	// Place to Basket 		
	4:
		IF process_Z = 0 THEN
			CASE GVL.Basket_A_Counter OF
				0:
					bit1 					:= 4;
					bit2 					:= 2;
					KR1.bOutBit[ bit1,bit2] := TRUE; //210
					MSG_Bskt				:= MSG.ACTION_FGA_POS1;
					process_Z 				:= 1;
				1:
					bit1 					:= 4;
					bit2 					:= 3;
					KR1.bOutBit[ bit1,bit2] := TRUE; //210
					MSG_Bskt				:= MSG.ACTION_FGA_POS2;
					process_Z 				:= 1;
					RETURN;
				2:
					bit1 					:= 4;
					bit2 					:= 4;
					KR1.bOutBit[ bit1,bit2] := TRUE; //210
					MSG_Bskt				:= MSG.ACTION_FGA_POS3;
					process_Z 				:= 1;
				3:
					bit1 					:= 4;
					bit2 					:= 5;
					KR1.bOutBit[ bit1,bit2] := TRUE; //210
					MSG_Bskt				:= MSG.ACTION_FGA_POS4;
					process_Z 				:= 1;
				4:
					bit1 					:= 4;
					bit2 					:= 6;
					KR1.bOutBit[ bit1,bit2] := TRUE; //210
					MSG_Bskt				:= MSG.ACTION_FGA_POS5;
					process_Z 				:= 1;
				5:
					bit1 					:= 4;
					bit2 					:= 7;
					KR1.bOutBit[ bit1,bit2] := TRUE; //210
					MSG_Bskt				:= MSG.ACTION_FGA_POS6;
					process_Z 				:= 1;
				6:
					bit1 					:= 5;
					bit2 					:= 0;
					KR1.bOutBit[ bit1,bit2] := TRUE; //210
					MSG_Bskt				:= MSG.ACTION_FGA_POS7;
					process_Z 				:= 1;
				7:
					bit1 					:= 5;
					bit2 					:= 1;
					KR1.bOutBit[ bit1,bit2] := TRUE; //210
					MSG_Bskt				:= MSG.ACTION_FGA_POS8;
					process_Z 				:= 1;
				8:
					bit1 					:= 5;
					bit2 					:= 2;
					KR1.bOutBit[ bit1,bit2] := TRUE; //210
					MSG_Bskt				:= MSG.ACTION_FGA_POS9;
					process_Z 				:= 1;
				9:
					bit1 					:= 5;
					bit2 					:= 3;
					KR1.bOutBit[ bit1,bit2] := TRUE; //210
					MSG_Bskt				:= MSG.ACTION_FGA_POS10;
					process_Z 				:= 1;
				10:
					bit1 					:= 5;
					bit2 					:= 4;
					KR1.bOutBit[ bit1,bit2] := TRUE; //210
					MSG_Bskt				:= MSG.ACTION_FGA_POS11;
					process_Z 				:= 1;
				11:
					bit1 					:= 5;
					bit2 					:= 5;
					KR1.bOutBit[ bit1,bit2] := TRUE; //210
					MSG_Bskt				:= MSG.ACTION_FGA_POS12;
					process_Z 				:= 1;
				12:
					bit1 					:= 5;
					bit2 					:= 6;
					KR1.bOutBit[ bit1,bit2] := TRUE; //210
					MSG_Bskt				:= MSG.ACTION_FGA_POS13;
					process_Z 				:= 1;
				13:
					bit1 					:= 5;
					bit2 					:= 7;
					KR1.bOutBit[ bit1,bit2] := TRUE; //210
					MSG_Bskt				:= MSG.ACTION_FGA_POS14;
					process_Z 				:= 1;
				14:
					bit1 					:= 6;
					bit2 					:= 0;
					KR1.bOutBit[ bit1,bit2] := TRUE; //210
					MSG_Bskt				:= MSG.ACTION_FGA_POS15;
					process_Z 				:= 1;
				15:
					bit1 					:= 6;
					bit2 					:= 1;
					KR1.bOutBit[ bit1,bit2] := TRUE; //210
					MSG_Bskt				:= MSG.ACTION_FGA_POS16;
					process_Z 				:= 1;
				16:
					bit1 					:= 6;
					bit2 					:= 2;
					KR1.bOutBit[ bit1,bit2] := TRUE; //210
					MSG_Bskt				:= MSG.ACTION_FGA_POS17;
					process_Z 				:= 1;
				17:
					bit1 					:= 6;
					bit2 					:= 3;
					KR1.bOutBit[ bit1,bit2] := TRUE; //210
					MSG_Bskt				:= MSG.ACTION_FGA_POS18;
					process_Z 				:= 1;
				18:
					bit1 					:= 6;
					bit2 					:= 4;
					KR1.bOutBit[ bit1,bit2] := TRUE; //210
					MSG_Bskt				:= MSG.ACTION_FGA_POS19;
					process_Z 				:= 1;
				19:
					bit1 					:= 6;
					bit2 					:= 5;
					KR1.bOutBit[ bit1,bit2] := TRUE; //210
					MSG_Bskt				:= MSG.ACTION_FGA_POS20;
					process_Z 				:= 1;
				20:
					bit1 					:= 6;
					bit2 					:= 6;
					KR1.bOutBit[ bit1,bit2] := TRUE; //210
					MSG_Bskt				:= MSG.ACTION_FGA_POS21;
					process_Z 				:= 1;
				21:
					bit1 					:= 6;
					bit2 					:= 7;
					KR1.bOutBit[ bit1,bit2] := TRUE; //210
					MSG_Bskt				:= MSG.ACTION_FGA_POS22;
					process_Z 				:= 1;
				22:
					bit1 					:= 7;
					bit2 					:= 0;
					KR1.bOutBit[ bit1,bit2] := TRUE; //210
					MSG_Bskt				:= MSG.ACTION_FGA_POS23;
					process_Z 				:= 1;
				23:
					bit1 					:= 7;
					bit2 					:= 1;
					KR1.bOutBit[ bit1,bit2] := TRUE; //210
					MSG_Bskt				:= MSG.ACTION_FGA_POS24;
					process_Z 				:= 1;
				24:
					bit1 					:= 7;
					bit2 					:= 2;
					KR1.bOutBit[ bit1,bit2] := TRUE; //210
					MSG_Bskt				:= MSG.ACTION_FGA_POS25;
					process_Z 				:= 1;
				25:
					bit1 					:= 7;
					bit2 					:= 3;
					KR1.bOutBit[ bit1,bit2] := TRUE; //210
					MSG_Bskt				:= MSG.ACTION_FGA_POS26;
					process_Z 				:= 1;
				26:
					bit1 					:= 7;
					bit2 					:= 4;
					KR1.bOutBit[ bit1,bit2] := TRUE; //210
					MSG_Bskt				:= MSG.ACTION_FGA_POS27;
					process_Z 				:= 1;
				27:
					bit1 					:= 7;
					bit2 					:= 5;
					KR1.bOutBit[ bit1,bit2] := TRUE; //210
					MSG_Bskt				:= MSG.ACTION_FGA_POS28;
					process_Z 				:= 1;
				28:
					bit1 					:= 7;
					bit2 					:= 6;
					KR1.bOutBit[ bit1,bit2] := TRUE; //210
					MSG_Bskt				:= MSG.ACTION_FGA_POS29;
					process_Z 				:= 1;
				29:
					bit1 					:= 7;
					bit2 					:= 7;
					KR1.bOutBit[ bit1,bit2] := TRUE; //210
					MSG_Bskt				:= MSG.ACTION_FGA_POS30;
					process_Z 				:= 1;
				30:
					bit1 					:= 8;
					bit2 					:= 0;
					KR1.bOutBit[ bit1,bit2] := TRUE; //210
					MSG_Bskt				:= MSG.ACTION_FGA_POS31;
					process_Z 				:= 1;
				31:
					bit1 					:= 8;
					bit2 					:= 1;
					KR1.bOutBit[ bit1,bit2] := TRUE; //210
					MSG_Bskt				:= MSG.ACTION_FGA_POS32;
					process_Z 				:= 1;
				32:
					bit1 					:= 8;
					bit2 					:= 2;
					KR1.bOutBit[ bit1,bit2] := TRUE; //210
					MSG_Bskt				:= MSG.ACTION_FGA_POS33;
					process_Z 				:= 1;
				33:
					bit1 					:= 8;
					bit2 					:= 3;
					KR1.bOutBit[ bit1,bit2] := TRUE; //210
					MSG_Bskt				:= MSG.ACTION_FGA_POS34;
					process_Z 				:= 1;
				34:
					bit1 					:= 8;
					bit2 					:= 4;
					KR1.bOutBit[ bit1,bit2] := TRUE; //210
					MSG_Bskt				:= MSG.ACTION_FGA_POS35;
					process_Z 				:= 1;
				35:
					bit1 					:= 8;
					bit2 					:= 5;
					KR1.bOutBit[ bit1,bit2] := TRUE; //210
					MSG_Bskt				:= MSG.ACTION_FGA_POS36;
					process_Z 				:= 1;
				36:
					bit1 					:= 8;
					bit2 					:= 6;
					KR1.bOutBit[ bit1,bit2] := TRUE; //210
					MSG_Bskt				:= MSG.ACTION_FGA_POS37;
					process_Z 				:= 1;
				37:
					bit1 					:= 8;
					bit2 					:= 7;
					KR1.bOutBit[ bit1,bit2] := TRUE; //210
					MSG_Bskt				:= MSG.ACTION_FGA_POS38;
					process_Z 				:= 1;
				38:
					bit1 					:= 9;
					bit2 					:= 0;
					KR1.bOutBit[ bit1,bit2] := TRUE; //210
					MSG_Bskt				:= MSG.ACTION_FGA_POS39;
					process_Z 				:= 1;
				39:
					bit1 					:= 9;
					bit2 					:= 1;
					KR1.bOutBit[ bit1,bit2] := TRUE; //210
					MSG_Bskt				:= MSG.ACTION_FGA_POS40;
					process_Z 				:= 1;
				40:
					bit1 					:= 9;
					bit2 					:= 2;
					KR1.bOutBit[ bit1,bit2] := TRUE; //210
					MSG_Bskt				:= MSG.ACTION_FGA_POS41;
					process_Z 				:= 1;
				41:
					bit1 					:= 9;
					bit2 					:= 3;
					KR1.bOutBit[ bit1,bit2] := TRUE; //210
					MSG_Bskt				:= MSG.ACTION_FGA_POS42;
					process_Z 				:= 1;
				42:
					bit1 					:= 9;
					bit2 					:= 4;
					KR1.bOutBit[ bit1,bit2] := TRUE; //210
					MSG_Bskt				:= MSG.ACTION_FGA_POS43;
					process_Z 				:= 1;
				43:
					bit1 					:= 9;
					bit2 					:= 5;
					KR1.bOutBit[ bit1,bit2] := TRUE; //210
					MSG_Bskt				:= MSG.ACTION_FGA_POS44;
					process_Z 				:= 1;
				44:
					bit1 					:= 9;
					bit2 					:= 6;
					KR1.bOutBit[ bit1,bit2] := TRUE; //210
					MSG_Bskt				:= MSG.ACTION_FGA_POS45;
					process_Z 				:= 1;
				45:
					bit1 					:= 9;
					bit2 					:= 7;
					KR1.bOutBit[ bit1,bit2] := TRUE; //210
					MSG_Bskt				:= MSG.ACTION_FGA_POS46;
					process_Z 				:= 1;
				46:
					bit1 					:= 10;
					bit2 					:= 0;
					KR1.bOutBit[ bit1,bit2] := TRUE; //210
					MSG_Bskt				:= MSG.ACTION_FGA_POS47;
					process_Z 				:= 1;
				47:
					bit1 					:= 10;
					bit2 					:= 1;
					KR1.bOutBit[ bit1,bit2] := TRUE; //210
					MSG_Bskt				:= MSG.ACTION_FGA_POS48;
					process_Z 				:= 1;
				48:
					bit1 					:= 10;
					bit2 					:= 2;
					KR1.bOutBit[ bit1,bit2] := TRUE; //210
					MSG_Bskt				:= MSG.ACTION_FGA_POS49;
					process_Z 				:= 1;
				49:
					bit1 					:= 10;
					bit2 					:= 3;
					KR1.bOutBit[ bit1,bit2] := TRUE; //210
					MSG_Bskt				:= MSG.ACTION_FGA_POS50;
					process_Z 				:= 1;
				50:
					bit1 					:= 10;
					bit2 					:= 4;
					KR1.bOutBit[ bit1,bit2] := TRUE; //210
					MSG_Bskt				:= MSG.ACTION_FGA_POS51;
					process_Z 				:= 1;
				51:
					bit1 					:= 10;
					bit2 					:= 5;
					KR1.bOutBit[ bit1,bit2] := TRUE; //210
					MSG_Bskt				:= MSG.ACTION_FGA_POS52;
					process_Z 				:= 1;
				52:
					bit1 					:= 10;
					bit2 					:= 6;
					KR1.bOutBit[ bit1,bit2] := TRUE; //210
					MSG_Bskt				:= MSG.ACTION_FGA_POS53;
					process_Z 				:= 1;
				53:
					bit1 					:= 10;
					bit2 					:= 7;
					KR1.bOutBit[ bit1,bit2] := TRUE; //210
					MSG_Bskt				:= MSG.ACTION_FGA_POS54;
					process_Z 				:= 1;
				54:
					bit1 					:= 11;
					bit2 					:= 0;
					KR1.bOutBit[ bit1,bit2] := TRUE; //210
					MSG_Bskt				:= MSG.ACTION_FGA_POS55;
					process_Z 				:= 1;
				55:
					bit1 					:= 11;
					bit2 					:= 1;
					KR1.bOutBit[ bit1,bit2] := TRUE; //210
					MSG_Bskt				:= MSG.ACTION_FGA_POS56;
					process_Z 				:= 1;
				56:
					bit1 					:= 11;
					bit2 					:= 2;
					KR1.bOutBit[ bit1,bit2] := TRUE; //210
					MSG_Bskt				:= MSG.ACTION_FGA_POS57;
					process_Z 				:= 1;
				57:
					bit1 					:= 11;
					bit2 					:= 3;
					KR1.bOutBit[ bit1,bit2] := TRUE; //210
					MSG_Bskt				:= MSG.ACTION_FGA_POS58;
					process_Z 				:= 1;
				58:
					bit1 					:= 11;
					bit2 					:= 4;
					KR1.bOutBit[ bit1,bit2] := TRUE; //210
					MSG_Bskt				:= MSG.ACTION_FGA_POS59;
					process_Z 				:= 1;
				59:
					bit1 					:= 11;
					bit2 					:= 5;
					KR1.bOutBit[ bit1,bit2] := TRUE; //210
					MSG_Bskt				:= MSG.ACTION_FGA_POS60;
					process_Z 				:= 1;
				60:
					bit1 					:= 11;
					bit2 					:= 6;
					KR1.bOutBit[ bit1,bit2] := TRUE; //210
					MSG_Bskt				:= MSG.ACTION_FGA_POS61;
					process_Z 				:= 1;
				61:
					bit1 					:= 11;
					bit2 					:= 7;
					KR1.bOutBit[ bit1,bit2] := TRUE; //210
					MSG_Bskt				:= MSG.ACTION_FGA_POS62;
					process_Z 				:= 1;
				62:
					bit1 					:= 12;
					bit2 					:= 0;
					KR1.bOutBit[ bit1,bit2] := TRUE; //210
					MSG_Bskt				:= MSG.ACTION_FGA_POS63;
					process_Z 				:= 1;
				63:
					bit1 					:= 12;
					bit2 					:= 1;
					KR1.bOutBit[ bit1,bit2] := TRUE; //210
					MSG_Bskt				:= MSG.ACTION_FGA_POS64;
					process_Z 				:= 1;
				64:
					bit1 					:= 12;
					bit2 					:= 2;
					KR1.bOutBit[ bit1,bit2] := TRUE; //210
					MSG_Bskt				:= MSG.ACTION_FGA_POS65;
					process_Z 				:= 1;
				65:
					bit1 					:= 12;
					bit2 					:= 3;
					KR1.bOutBit[ bit1,bit2] := TRUE; //210
					MSG_Bskt				:= MSG.ACTION_FGA_POS66;
					process_Z 				:= 1;
				66:
					bit1 					:= 12;
					bit2 					:= 4;
					KR1.bOutBit[ bit1,bit2] := TRUE; //210
					MSG_Bskt				:= MSG.ACTION_FGA_POS67;
					process_Z 				:= 1;
				67:
					bit1 					:= 12;
					bit2 					:= 5;
					KR1.bOutBit[ bit1,bit2] := TRUE; //210
					MSG_Bskt				:= MSG.ACTION_FGA_POS68;
					process_Z 				:= 1;
				68:
					bit1 					:= 12;
					bit2 					:= 6;
					KR1.bOutBit[ bit1,bit2] := TRUE; //210
					MSG_Bskt				:= MSG.ACTION_FGA_POS69;
					process_Z 				:= 1;
				69:
					bit1 					:= 12;
					bit2 					:= 7;
					KR1.bOutBit[ bit1,bit2] := TRUE; //210
					MSG_Bskt				:= MSG.ACTION_FGA_POS70;
					process_Z 				:= 1;
				70:
					bit1 					:= 13;
					bit2 					:= 0;
					KR1.bOutBit[ bit1,bit2] := TRUE; //210
					MSG_Bskt				:= MSG.ACTION_FGA_POS71;
					process_Z 				:= 1;
				71:
					bit1 					:= 13;
					bit2 					:= 1;
					KR1.bOutBit[ bit1,bit2] := TRUE; //210
					MSG_Bskt				:= MSG.ACTION_FGA_POS72;
					process_Z 				:= 1;
				72:
					bit1 					:= 13;
					bit2 					:= 2;
					KR1.bOutBit[ bit1,bit2] := TRUE; //210
					MSG_Bskt				:= MSG.ACTION_FGA_POS73;
					process_Z 				:= 1;
				73:
					bit1 					:= 13;
					bit2 					:= 3;
					KR1.bOutBit[ bit1,bit2] := TRUE; //210
					MSG_Bskt				:= MSG.ACTION_FGA_POS74;
					process_Z 				:= 1;
				74:
					bit1 					:= 13;
					bit2 					:= 4;
					KR1.bOutBit[ bit1,bit2] := TRUE; //210
					MSG_Bskt				:= MSG.ACTION_FGA_POS75;
					process_Z 				:= 1;
				75:
					bit1 					:= 13;
					bit2 					:= 5;
					KR1.bOutBit[ bit1,bit2] := TRUE; //210
					MSG_Bskt				:= MSG.ACTION_FGA_POS76;
					process_Z 				:= 1;
				76:
					bit1 					:= 13;
					bit2 					:= 6;
					KR1.bOutBit[ bit1,bit2] := TRUE; //210
					MSG_Bskt				:= MSG.ACTION_FGA_POS77;
					process_Z 				:= 1;
				77:
					bit1 					:= 13;
					bit2 					:= 7;
					KR1.bOutBit[ bit1,bit2] := TRUE; //210
					MSG_Bskt				:= MSG.ACTION_FGA_POS78;
					process_Z 				:= 1;
				78:
					bit1 					:= 14;
					bit2 					:= 0;
					KR1.bOutBit[ bit1,bit2] := TRUE; //210
					MSG_Bskt				:= MSG.ACTION_FGA_POS79;
					process_Z 				:= 1;
				79:
					bit1 					:= 14;
					bit2 					:= 1;
					KR1.bOutBit[ bit1,bit2] := TRUE; //210
					MSG_Bskt				:= MSG.ACTION_FGA_POS80;
					process_Z 				:= 1;
				80:
					bit1 					:= 14;
					bit2 					:= 2;
					KR1.bOutBit[ bit1,bit2] := TRUE; //210
					MSG_Bskt				:= MSG.ACTION_FGA_POS81;
					process_Z 				:= 1;
				81:
					bit1 					:= 14;
					bit2 					:= 3;
					KR1.bOutBit[ bit1,bit2] := TRUE; //210
					MSG_Bskt				:= MSG.ACTION_FGA_POS82;
					process_Z 				:= 1;
				82:
					bit1 					:= 14;
					bit2 					:= 4;
					KR1.bOutBit[ bit1,bit2] := TRUE; //210
					MSG_Bskt				:= MSG.ACTION_FGA_POS83;
					process_Z 				:= 1;
				83:
					bit1 					:= 14;
					bit2 					:= 5;
					KR1.bOutBit[ bit1,bit2] := TRUE; //210
					MSG_Bskt				:= MSG.ACTION_FGA_POS84;
					process_Z 				:= 1;
				84:
					bit1 					:= 14;
					bit2 					:= 6;
					KR1.bOutBit[ bit1,bit2] := TRUE; //210
					MSG_Bskt				:= MSG.ACTION_FGA_POS85;
					process_Z 				:= 1;
				85:
					bit1 					:= 14;
					bit2 					:= 7;
					KR1.bOutBit[ bit1,bit2] := TRUE; //210
					MSG_Bskt				:= MSG.ACTION_FGA_POS86;
					process_Z 				:= 1;
				86:
					bit1 					:= 15;
					bit2 					:= 0;
					KR1.bOutBit[ bit1,bit2] := TRUE; //210
					MSG_Bskt				:= MSG.ACTION_FGA_POS87;
					process_Z 				:= 1;
				87:
					bit1 					:= 15;
					bit2 					:= 1;
					KR1.bOutBit[ bit1,bit2] := TRUE; //210
					MSG_Bskt				:= MSG.ACTION_FGA_POS88;
					process_Z 				:= 1;
				88:
					bit1 					:= 15;
					bit2 					:= 2;
					KR1.bOutBit[ bit1,bit2] := TRUE; //210
					MSG_Bskt				:= MSG.ACTION_FGA_POS89;
					process_Z 				:= 1;
				89:
					bit1 					:= 15;
					bit2 					:= 3;
					KR1.bOutBit[ bit1,bit2] := TRUE; //210
					MSG_Bskt				:= MSG.ACTION_FGA_POS90;
					process_Z 				:= 1;
				90:
					bit1 					:= 15;
					bit2 					:= 4;
					KR1.bOutBit[ bit1,bit2] := TRUE; //210
					MSG_Bskt				:= MSG.ACTION_FGA_POS91;
					process_Z 				:= 1;
				91:
					bit1 					:= 15;
					bit2 					:= 5;
					KR1.bOutBit[ bit1,bit2] := TRUE; //210
					MSG_Bskt				:= MSG.ACTION_FGA_POS92;
					process_Z 				:= 1;
				92:
					bit1 					:= 15;
					bit2 					:= 6;
					KR1.bOutBit[ bit1,bit2] := TRUE; //210
					MSG_Bskt				:= MSG.ACTION_FGA_POS93;
					process_Z 				:= 1;
				93:
					bit1 					:= 15;
					bit2 					:= 7;
					KR1.bOutBit[ bit1,bit2] := TRUE; //210
					MSG_Bskt				:= MSG.ACTION_FGA_POS94;
					process_Z 				:= 1;
				94:
					bit1 					:= 16;
					bit2 					:= 0;
					KR1.bOutBit[ bit1,bit2] := TRUE; //210
					MSG_Bskt				:= MSG.ACTION_FGA_POS95;
					process_Z 				:= 1;
				95:
					bit1 					:= 16;
					bit2 					:= 1;
					KR1.bOutBit[ bit1,bit2] := TRUE; //210
					MSG_Bskt				:= MSG.ACTION_FGA_POS96;
					process_Z 				:= 1;
				96:
					bit1 					:= 16;
					bit2 					:= 2;
					KR1.bOutBit[ bit1,bit2] := TRUE; //210
					MSG_Bskt				:= MSG.ACTION_FGA_POS97;
					process_Z 				:= 1;
				97:
					bit1 					:= 16;
					bit2 					:= 3;
					KR1.bOutBit[ bit1,bit2] := TRUE; //210
					MSG_Bskt				:= MSG.ACTION_FGA_POS98;
					process_Z 				:= 1;
				98:
					bit1 					:= 16;
					bit2 					:= 4;
					KR1.bOutBit[ bit1,bit2] := TRUE; //210
					MSG_Bskt				:= MSG.ACTION_FGA_POS99;
					process_Z 				:= 1;
				99:
					bit1 					:= 16;
					bit2 					:= 5;
					KR1.bOutBit[ bit1,bit2] := TRUE; //210
					MSG_Bskt				:= MSG.ACTION_FGA_POS100;
					process_Z 				:= 1;
				100:
					bit1 					:= 16;
					bit2 					:= 6;
					KR1.bOutBit[ bit1,bit2] := TRUE; //210
					MSG_Bskt				:= MSG.ACTION_FGA_POS101;
					process_Z 				:= 1;
				101:
					bit1 					:= 16;
					bit2 					:= 7;
					KR1.bOutBit[ bit1,bit2] := TRUE; //210
					MSG_Bskt				:= MSG.ACTION_FGA_POS102;
					process_Z 				:= 1;
				102:
					bit1 					:= 17;
					bit2 					:= 0;
					KR1.bOutBit[ bit1,bit2] := TRUE; //210
					MSG_Bskt				:= MSG.ACTION_FGA_POS103;
					process_Z 				:= 1;
				103:
					bit1 					:= 17;
					bit2 					:= 1;
					KR1.bOutBit[ bit1,bit2] := TRUE; //210
					MSG_Bskt				:= MSG.ACTION_FGA_POS104;
					process_Z 				:= 1;
				104:
					bit1 					:= 17;
					bit2 					:= 2;
					KR1.bOutBit[ bit1,bit2] := TRUE; //210
					MSG_Bskt				:= MSG.ACTION_FGA_POS105;
					process_Z 				:= 1;
				105:
					bit1 					:= 17;
					bit2 					:= 3;
					KR1.bOutBit[ bit1,bit2] := TRUE; //210
					MSG_Bskt				:= MSG.ACTION_FGA_POS106;
					process_Z 				:= 1;
				106:
					bit1 					:= 17;
					bit2 					:= 4;
					KR1.bOutBit[ bit1,bit2] := TRUE; //210
					MSG_Bskt				:= MSG.ACTION_FGA_POS107;
					process_Z 				:= 1;
				107:
					bit1 					:= 17;
					bit2 					:= 5;
					KR1.bOutBit[ bit1,bit2] := TRUE; //210
					MSG_Bskt				:= MSG.ACTION_FGA_POS108;
					process_Z 				:= 1;
				108:
					bit1 					:= 17;
					bit2 					:= 6;
					KR1.bOutBit[ bit1,bit2] := TRUE; //210
					MSG_Bskt				:= MSG.ACTION_FGA_POS109;
					process_Z 				:= 1;
				109:
					bit1 					:= 17;
					bit2 					:= 7;
					KR1.bOutBit[ bit1,bit2] := TRUE; //210
					MSG_Bskt				:= MSG.ACTION_FGA_POS110;
					process_Z 				:= 1;
				110:
					bit1 					:= 18;
					bit2 					:= 0;
					KR1.bOutBit[ bit1,bit2] := TRUE; //210
					MSG_Bskt				:= MSG.ACTION_FGA_POS111;
					process_Z 				:= 1;
				111:
					bit1 					:= 18;
					bit2 					:= 1;
					KR1.bOutBit[ bit1,bit2] := TRUE; //210
					MSG_Bskt				:= MSG.ACTION_FGA_POS112;
					process_Z 				:= 1;
				112:
					bit1 					:= 18;
					bit2 					:= 2;
					KR1.bOutBit[ bit1,bit2] := TRUE; //210
					MSG_Bskt				:= MSG.ACTION_FGA_POS113;
					process_Z 				:= 1;
				113:
					bit1 					:= 18;
					bit2 					:= 3;
					KR1.bOutBit[ bit1,bit2] := TRUE; //210
					MSG_Bskt				:= MSG.ACTION_FGA_POS114;
					process_Z 				:= 1;
				114:
					bit1 					:= 18;
					bit2 					:= 4;
					KR1.bOutBit[ bit1,bit2] := TRUE; //210
					MSG_Bskt				:= MSG.ACTION_FGA_POS115;
					process_Z 				:= 1;
				115:
					bit1 					:= 18;
					bit2 					:= 5;
					KR1.bOutBit[ bit1,bit2] := TRUE; //210
					MSG_Bskt				:= MSG.ACTION_FGA_POS116;
					process_Z 				:= 1;
				116:
					bit1 					:= 18;
					bit2 					:= 6;
					KR1.bOutBit[ bit1,bit2] := TRUE; //210
					MSG_Bskt				:= MSG.ACTION_FGA_POS117;
					process_Z 				:= 1;
				117:
					bit1 					:= 18;
					bit2 					:= 7;
					KR1.bOutBit[ bit1,bit2] := TRUE; //210
					MSG_Bskt				:= MSG.ACTION_FGA_POS118;
					process_Z 				:= 1;
				118:
					bit1 					:= 19;
					bit2 					:= 0;
					KR1.bOutBit[ bit1,bit2] := TRUE; //210
					MSG_Bskt				:= MSG.ACTION_FGA_POS119;
					process_Z 				:= 1;
				119:
					bit1 					:= 19;
					bit2 					:= 1;
					KR1.bOutBit[ bit1,bit2] := TRUE; //210
					MSG_Bskt				:= MSG.ACTION_FGA_POS120;
					process_Z 				:= 1;
				120:
					bit1 					:= 19;
					bit2 					:= 2;
					KR1.bOutBit[ bit1,bit2] := TRUE; //210
					MSG_Bskt				:= MSG.ACTION_FGA_POS121;
					process_Z 				:= 1;
				121:
					bit1 					:= 19;
					bit2 					:= 3;
					KR1.bOutBit[ bit1,bit2] := TRUE; //210
					MSG_Bskt				:= MSG.ACTION_FGA_POS122;
					process_Z 				:= 1;
				122:
					bit1 					:= 19;
					bit2 					:= 4;
					KR1.bOutBit[ bit1,bit2] := TRUE; //210
					MSG_Bskt				:= MSG.ACTION_FGA_POS123;
					process_Z 				:= 1;
				123:
					bit1 					:= 19;
					bit2 					:= 5;
					KR1.bOutBit[ bit1,bit2] := TRUE; //210
					MSG_Bskt				:= MSG.ACTION_FGA_POS124;
					process_Z 				:= 1;
				124:
					bit1 					:= 19;
					bit2 					:= 6;
					KR1.bOutBit[ bit1,bit2] := TRUE; //210
					MSG_Bskt				:= MSG.ACTION_FGA_POS125;
					process_Z 				:= 1;
				125:
					bit1 					:= 19;
					bit2 					:= 7;
					KR1.bOutBit[ bit1,bit2] := TRUE; //210
					MSG_Bskt				:= MSG.ACTION_FGA_POS126;
					process_Z 				:= 1;
				126:
					bit1 					:= 20;
					bit2 					:= 0;
					KR1.bOutBit[ bit1,bit2] := TRUE; //210
					MSG_Bskt				:= MSG.ACTION_FGA_POS127;
					process_Z 				:= 1;
				127:
					bit1 					:= 20;
					bit2 					:= 1;
					KR1.bOutBit[ bit1,bit2] := TRUE; //210
					MSG_Bskt				:= MSG.ACTION_FGA_POS128;
					process_Z 				:= 1;
				128:
					bit1 					:= 20;
					bit2 					:= 2;
					KR1.bOutBit[ bit1,bit2] := TRUE; //210
					MSG_Bskt				:= MSG.ACTION_FGA_POS129;
					process_Z 				:= 1;
				129:
					bit1 					:= 20;
					bit2 					:= 3;
					KR1.bOutBit[ bit1,bit2] := TRUE; //210
					MSG_Bskt				:= MSG.ACTION_FGA_POS130;
					process_Z 				:= 1;
				130:
					bit1 					:= 20;
					bit2 					:= 4;
					KR1.bOutBit[ bit1,bit2] := TRUE; //210
					MSG_Bskt				:= MSG.ACTION_FGA_POS131;
					process_Z 				:= 1;
				131:
					bit1 					:= 20;
					bit2 					:= 5;
					KR1.bOutBit[ bit1,bit2] := TRUE; //210
					MSG_Bskt				:= MSG.ACTION_FGA_POS132;
					process_Z 				:= 1;
				132:
					bit1 					:= 20;
					bit2 					:= 6;
					KR1.bOutBit[ bit1,bit2] := TRUE; //210
					MSG_Bskt				:= MSG.ACTION_FGA_POS133;
					process_Z 				:= 1;
				133:
					bit1 					:= 20;
					bit2 					:= 7;
					KR1.bOutBit[ bit1,bit2] := TRUE; //210
					MSG_Bskt				:= MSG.ACTION_FGA_POS134;
					process_Z 				:= 1;
				134:
					bit1 					:= 21;
					bit2 					:= 0;
					KR1.bOutBit[ bit1,bit2] := TRUE; //210
					MSG_Bskt				:= MSG.ACTION_FGA_POS135;
					process_Z 				:= 1;
				135:
					bit1 					:= 21;
					bit2 					:= 1;
					KR1.bOutBit[ bit1,bit2] := TRUE; //210
					MSG_Bskt				:= MSG.ACTION_FGA_POS136;
					process_Z 				:= 1;
				136:
					bit1 					:= 21;
					bit2 					:= 2;
					KR1.bOutBit[ bit1,bit2] := TRUE; //210
					MSG_Bskt				:= MSG.ACTION_FGA_POS137;
					process_Z 				:= 1;
				137:
					bit1 					:= 21;
					bit2 					:= 3;
					KR1.bOutBit[ bit1,bit2] := TRUE; //210
					MSG_Bskt				:= MSG.ACTION_FGA_POS138;
					process_Z 				:= 1;
				138:
					bit1 					:= 21;
					bit2 					:= 4;
					KR1.bOutBit[ bit1,bit2] := TRUE; //210
					MSG_Bskt				:= MSG.ACTION_FGA_POS139;
					process_Z 				:= 1;
				139:
					bit1 					:= 21;
					bit2 					:= 5;
					KR1.bOutBit[ bit1,bit2] := TRUE; //210
					MSG_Bskt				:= MSG.ACTION_FGA_POS140;
					process_Z 				:= 1;
				140:
					bit1 					:= 21;
					bit2 					:= 6;
					KR1.bOutBit[ bit1,bit2] := TRUE; //210
					MSG_Bskt				:= MSG.ACTION_FGA_POS141;
					process_Z 				:= 1;
				141:
					bit1 					:= 21;
					bit2 					:= 7;
					KR1.bOutBit[ bit1,bit2] := TRUE; //210
					MSG_Bskt				:= MSG.ACTION_FGA_POS142;
					process_Z 				:= 1;
				142:
					bit1 					:= 22;
					bit2 					:= 0;
					KR1.bOutBit[ bit1,bit2] := TRUE; //210
					MSG_Bskt				:= MSG.ACTION_FGA_POS143;
					process_Z 				:= 1;
				143:
					bit1 					:= 22;
					bit2 					:= 1;
					KR1.bOutBit[ bit1,bit2] := TRUE; //210
					MSG_Bskt				:= MSG.ACTION_FGA_POS144;
					process_Z 				:= 1;
				144:
					bit1 					:= 22;
					bit2 					:= 2;
					KR1.bOutBit[ bit1,bit2] := TRUE; //210
					MSG_Bskt				:= MSG.ACTION_FGA_POS145;
					process_Z 				:= 1;
				145:
					bit1 					:= 22;
					bit2 					:= 3;
					KR1.bOutBit[ bit1,bit2] := TRUE; //210
					MSG_Bskt				:= MSG.ACTION_FGA_POS146;
					process_Z 				:= 1;
				146:
					bit1 					:= 22;
					bit2 					:= 4;
					KR1.bOutBit[ bit1,bit2] := TRUE; //210
					MSG_Bskt				:= MSG.ACTION_FGA_POS147;
					process_Z 				:= 1;
				147:
					bit1 					:= 22;
					bit2 					:= 5;
					KR1.bOutBit[ bit1,bit2] := TRUE; //210
					MSG_Bskt				:= MSG.ACTION_FGA_POS148;
					process_Z 				:= 1;
				148:
					bit1 					:= 22;
					bit2 					:= 6;
					KR1.bOutBit[ bit1,bit2] := TRUE; //210
					MSG_Bskt				:= MSG.ACTION_FGA_POS149;
					process_Z 				:= 1;
				149:
					bit1 					:= 22;
					bit2 					:= 7;
					KR1.bOutBit[ bit1,bit2] := TRUE; //210
					MSG_Bskt				:= MSG.ACTION_FGA_POS150;
					process_Z 				:= 1;
				150:
					bit1 					:= 23;
					bit2 					:= 0;
					KR1.bOutBit[ bit1,bit2] := TRUE; //210
					MSG_Bskt				:= MSG.ACTION_FGA_POS151;
					process_Z 				:= 1;
				151:
					bit1 					:= 23;
					bit2 					:= 1;
					KR1.bOutBit[ bit1,bit2] := TRUE; //210
					MSG_Bskt				:= MSG.ACTION_FGA_POS152;
					process_Z 				:= 1;
				152:
					bit1 					:= 23;
					bit2 					:= 2;
					KR1.bOutBit[ bit1,bit2] := TRUE; //210
					MSG_Bskt				:= MSG.ACTION_FGA_POS153;
					process_Z 				:= 1;
				153:
					bit1 					:= 23;
					bit2 					:= 3;
					KR1.bOutBit[ bit1,bit2] := TRUE; //210
					MSG_Bskt				:= MSG.ACTION_FGA_POS154;
					process_Z 				:= 1;
				154:
					bit1 					:= 23;
					bit2 					:= 4;
					KR1.bOutBit[ bit1,bit2] := TRUE; //210
					MSG_Bskt				:= MSG.ACTION_FGA_POS155;
					process_Z 				:= 1;
				155:
					bit1 					:= 23;
					bit2 					:= 5;
					KR1.bOutBit[ bit1,bit2] := TRUE; //210
					MSG_Bskt				:= MSG.ACTION_FGA_POS156;
					process_Z 				:= 1;
				156:
					bit1 					:= 23;
					bit2 					:= 6;
					KR1.bOutBit[ bit1,bit2] := TRUE; //210
					MSG_Bskt				:= MSG.ACTION_FGA_POS157;
					process_Z 				:= 1;
				157:
					bit1 					:= 23;
					bit2 					:= 7;
					KR1.bOutBit[ bit1,bit2] := TRUE; //210
					MSG_Bskt				:= MSG.ACTION_FGA_POS158;
					process_Z 				:= 1;
				158:
					bit1 					:= 24;
					bit2 					:= 0;
					KR1.bOutBit[ bit1,bit2] := TRUE; //210
					MSG_Bskt				:= MSG.ACTION_FGA_POS159;
					process_Z 				:= 1;
				159:
					bit1 					:= 24;
					bit2 					:= 1;
					KR1.bOutBit[ bit1,bit2] := TRUE; //210
					MSG_Bskt				:= MSG.ACTION_FGA_POS160;
					process_Z 				:= 1;
				160:
					bit1 					:= 24;
					bit2 					:= 2;
					KR1.bOutBit[ bit1,bit2] := TRUE; //210
					MSG_Bskt				:= MSG.ACTION_FGA_POS161;
					process_Z 				:= 1;
				161:
					bit1 					:= 24;
					bit2 					:= 3;
					KR1.bOutBit[ bit1,bit2] := TRUE; //210
					MSG_Bskt				:= MSG.ACTION_FGA_POS162;
					process_Z 				:= 1;
				162:
					bit1 					:= 24;
					bit2 					:= 4;
					KR1.bOutBit[ bit1,bit2] := TRUE; //210
					MSG_Bskt				:= MSG.ACTION_FGA_POS163;
					process_Z 				:= 1;
				163:
					bit1 					:= 24;
					bit2 					:= 5;
					KR1.bOutBit[ bit1,bit2] := TRUE; //210
					MSG_Bskt				:= MSG.ACTION_FGA_POS164;
					process_Z 				:= 1;
				164:
					bit1 					:= 24;
					bit2 					:= 6;
					KR1.bOutBit[ bit1,bit2] := TRUE; //210
					MSG_Bskt				:= MSG.ACTION_FGA_POS165;
					process_Z 				:= 1;
				165:
					bit1 					:= 24;
					bit2 					:= 7;
					KR1.bOutBit[ bit1,bit2] := TRUE; //210
					MSG_Bskt				:= MSG.ACTION_FGA_POS166;
					process_Z 				:= 1;
				166:
					bit1 					:= 25;
					bit2 					:= 0;
					KR1.bOutBit[ bit1,bit2] := TRUE; //210
					MSG_Bskt				:= MSG.ACTION_FGA_POS167;
					process_Z 				:= 1;
				167:
					bit1 					:= 25;
					bit2 					:= 1;
					KR1.bOutBit[ bit1,bit2] := TRUE; //210
					MSG_Bskt				:= MSG.ACTION_FGA_POS168;
					process_Z 				:= 1;
				168:
					bit1 					:= 25;
					bit2 					:= 2;
					KR1.bOutBit[ bit1,bit2] := TRUE; //210
					MSG_Bskt				:= MSG.ACTION_FGA_POS169;
					process_Z 				:= 1;
				169:
					bit1 					:= 25;
					bit2 					:= 3;
					KR1.bOutBit[ bit1,bit2] := TRUE; //210
					MSG_Bskt				:= MSG.ACTION_FGA_POS170;
					process_Z 				:= 1;
				170:
					bit1 					:= 25;
					bit2 					:= 4;
					KR1.bOutBit[ bit1,bit2] := TRUE; //210
					MSG_Bskt				:= MSG.ACTION_FGA_POS171;
					process_Z 				:= 1;
				171:
					bit1 					:= 25;
					bit2 					:= 5;
					KR1.bOutBit[ bit1,bit2] := TRUE; //210
					MSG_Bskt				:= MSG.ACTION_FGA_POS172;
					process_Z 				:= 1;
				172:
					bit1 					:= 25;
					bit2 					:= 6;
					KR1.bOutBit[ bit1,bit2] := TRUE; //210
					MSG_Bskt				:= MSG.ACTION_FGA_POS173;
					process_Z 				:= 1;
				173:
					bit1 					:= 25;
					bit2 					:= 7;
					KR1.bOutBit[ bit1,bit2] := TRUE; //210
					MSG_Bskt				:= MSG.ACTION_FGA_POS174;
					process_Z 				:= 1;
				174:
					bit1 					:= 26;
					bit2 					:= 0;
					KR1.bOutBit[ bit1,bit2] := TRUE; //210
					MSG_Bskt				:= MSG.ACTION_FGA_POS175;
					process_Z 				:= 1;
				175:
					bit1 					:= 26;
					bit2 					:= 1;
					KR1.bOutBit[ bit1,bit2] := TRUE; //210
					MSG_Bskt				:= MSG.ACTION_FGA_POS176;
					process_Z 				:= 1;
				176:
					bit1 					:= 26;
					bit2 					:= 2;
					KR1.bOutBit[ bit1,bit2] := TRUE; //210
					MSG_Bskt				:= MSG.ACTION_FGA_POS177;
					process_Z 				:= 1;
				177:
					bit1 					:= 26;
					bit2 					:= 3;
					KR1.bOutBit[ bit1,bit2] := TRUE; //210
					MSG_Bskt				:= MSG.ACTION_FGA_POS178;
					process_Z 				:= 1;
				178:
					bit1 					:= 26;
					bit2 					:= 4;
					KR1.bOutBit[ bit1,bit2] := TRUE; //210
					MSG_Bskt				:= MSG.ACTION_FGA_POS179;
					process_Z 				:= 1;
				179:
					bit1 					:= 26;
					bit2 					:= 5;
					KR1.bOutBit[ bit1,bit2] := TRUE; //210
					MSG_Bskt				:= MSG.ACTION_FGA_POS180;
					process_Z 				:= 1;
				180:
					bit1 					:= 26;
					bit2 					:= 6;
					KR1.bOutBit[ bit1,bit2] := TRUE; //210
					MSG_Bskt				:= MSG.ACTION_FGA_POS181;
					process_Z 				:= 1;
				181:
					bit1 					:= 26;
					bit2 					:= 7;
					KR1.bOutBit[ bit1,bit2] := TRUE; //210
					MSG_Bskt				:= MSG.ACTION_FGA_POS182;
					process_Z 				:= 1;
				182:
					bit1 					:= 27;
					bit2 					:= 0;
					KR1.bOutBit[ bit1,bit2] := TRUE; //210
					MSG_Bskt				:= MSG.ACTION_FGA_POS183;
					process_Z 				:= 1;
				183:
					bit1 					:= 27;
					bit2 					:= 1;
					KR1.bOutBit[ bit1,bit2] := TRUE; //210
					MSG_Bskt				:= MSG.ACTION_FGA_POS184;
					process_Z 				:= 1;
				184:
					bit1 					:= 27;
					bit2 					:= 2;
					KR1.bOutBit[ bit1,bit2] := TRUE; //210
					MSG_Bskt				:= MSG.ACTION_FGA_POS185;
					process_Z 				:= 1;
				185:
					bit1 					:= 27;
					bit2 					:= 3;
					KR1.bOutBit[ bit1,bit2] := TRUE; //210
					MSG_Bskt				:= MSG.ACTION_FGA_POS186;
					process_Z 				:= 1;
				186:
					bit1 					:= 27;
					bit2 					:= 4;
					KR1.bOutBit[ bit1,bit2] := TRUE; //210
					MSG_Bskt				:= MSG.ACTION_FGA_POS187;
					process_Z 				:= 1;
				187:
					bit1 					:= 27;
					bit2 					:= 5;
					KR1.bOutBit[ bit1,bit2] := TRUE; //210
					MSG_Bskt				:= MSG.ACTION_FGA_POS188;
					process_Z 				:= 1;
				188:
					bit1 					:= 27;
					bit2 					:= 6;
					KR1.bOutBit[ bit1,bit2] := TRUE; //210
					MSG_Bskt				:= MSG.ACTION_FGA_POS189;
					process_Z 				:= 1;
				189:
					bit1 					:= 27;
					bit2 					:= 7;
					KR1.bOutBit[ bit1,bit2] := TRUE; //210
					MSG_Bskt				:= MSG.ACTION_FGA_POS190;
					process_Z 				:= 1;
				190:
					bit1 					:= 28;
					bit2 					:= 0;
					KR1.bOutBit[ bit1,bit2] := TRUE; //210
					MSG_Bskt				:= MSG.ACTION_FGA_POS191;
					process_Z 				:= 1;
				191:
					bit1 					:= 28;
					bit2 					:= 1;
					KR1.bOutBit[ bit1,bit2] := TRUE; //210
					MSG_Bskt				:= MSG.ACTION_FGA_POS192;
					process_Z 				:= 1;
				192:
					bit1 					:= 28;
					bit2 					:= 2;
					KR1.bOutBit[ bit1,bit2] := TRUE; //210
					MSG_Bskt				:= MSG.ACTION_FGA_POS193;
					process_Z 				:= 1;
				193:
					bit1 					:= 28;
					bit2 					:= 3;
					KR1.bOutBit[ bit1,bit2] := TRUE; //210
					MSG_Bskt				:= MSG.ACTION_FGA_POS194;
					process_Z 				:= 1;
				194:
					bit1 					:= 28;
					bit2 					:= 4;
					KR1.bOutBit[ bit1,bit2] := TRUE; //210
					MSG_Bskt				:= MSG.ACTION_FGA_POS195;
					process_Z 				:= 1;
				195:
					bit1 					:= 28;
					bit2 					:= 5;
					KR1.bOutBit[ bit1,bit2] := TRUE; //210
					MSG_Bskt				:= MSG.ACTION_FGA_POS196;
					process_Z 				:= 1;
				196:
					bit1 					:= 28;
					bit2 					:= 6;
					KR1.bOutBit[ bit1,bit2] := TRUE; //210
					MSG_Bskt				:= MSG.ACTION_FGA_POS197;
					process_Z 				:= 1;
				197:
					bit1 					:= 28;
					bit2 					:= 7;
					KR1.bOutBit[ bit1,bit2] := TRUE; //210
					MSG_Bskt				:= MSG.ACTION_FGA_POS198;
					process_Z 				:= 1;
				198:
					bit1 					:= 29;
					bit2 					:= 0;
					KR1.bOutBit[ bit1,bit2] := TRUE; //210
					MSG_Bskt				:= MSG.ACTION_FGA_POS199;
					process_Z 				:= 1;
				199:
					bit1 					:= 29;
					bit2 					:= 1;
					KR1.bOutBit[ bit1,bit2] := TRUE; //210
					MSG_Bskt				:= MSG.ACTION_FGA_POS200;
					process_Z 				:= 1;
			END_CASE
			AUTO_MODE.processnameFG := CONCAT(MSG.COMP_FG,MSG_Bskt);
			AUTO_MODE.processnameFG := CONCAT(AUTO_MODE.processnameFG,MSG.STATUS_RUN);
			LOGPROCESS( spLogComp	 := MSG.COMP_FG, 
						spLogAction	 := MSG_Bskt, 
						spLogStatus	 := MSG.STATUS_RUN,
						plogFlag	 := TRUE);
		ELSIF process_Z = 1 THEN
			KR1.bOutBit[ bit1,bit2] := TRUE;
			IF KR1.bInBit[ bit1,bit2] THEN
				KR1.bOutBit[ bit1,bit2] := FALSE;
				AUTO_MODE.processnameFG := CONCAT(MSG.COMP_FG,MSG.ACTION_FGA_POS);
				AUTO_MODE.processnameFG := CONCAT(AUTO_MODE.processnameFG,MSG.STATUS_ACK);
				LOGPROCESS( spLogComp	 := MSG.COMP_FG, 
							spLogAction	 := MSG.ACTION_FGA_POS, 
							spLogStatus	 := MSG.STATUS_ACK,
							plogFlag	 := TRUE);
				process_Z := 2;
				RETURN;
			END_IF	
		ELSIF process_Z = 2 THEN
			KR1.bOutBit[ bit1,bit2] := FALSE;
			IF NOT KR1.bInBit[ bit1,bit2] THEN
				AUTO_MODE.processnameFG := CONCAT(MSG.COMP_FG,MSG.ACTION_FGA_POS);
				AUTO_MODE.processnameFG := CONCAT(AUTO_MODE.processnameFG,MSG.STATUS_DONE);
				LOGPROCESS( spLogComp	 := MSG.COMP_FG, 
							spLogAction	 := MSG.ACTION_FGA_POS, 
							spLogStatus	 := MSG.STATUS_DONE,
							plogFlag	 := TRUE);
				process_Z:= 3;
				GVL.daily_output := GVL.daily_output+1;
				GVL.weekly_output := GVL.weekly_output+1;
				GVL.monthly_output := GVL.monthly_output+1;
				
				IF GVL.Basket_A_Counter < 15 THEN
					GVL.Basket_A_Counter := GVL.Basket_A_Counter+1;
				ELSE
					GVL.Basket_A_Counter := 0;
				END_IF
				
				FG_sequence := 5;
				AUTO_MODE.next_step := FALSE;
				AUTO_MODE.RW_PACKING := FALSE;
				AUTO_MODE.processnameFG := CONCAT(MSG.COMP_FG,MSG.ACTION_FGA_POS);
				AUTO_MODE.processnameFG := CONCAT(AUTO_MODE.processnameFG,MSG.STATUS_COMP);
				LOGPROCESS( spLogComp	 := MSG.COMP_FG, 
							spLogAction	 := MSG.ACTION_FGA_POS, 
							spLogStatus	 := MSG.STATUS_COMP,
							plogFlag	 := TRUE);
			END_IF	
		END_IF
		
	5:
		IF GVL.Basket_A_Counter = 15 THEN
			fb_RunLayerPad(Basket := 1, Layer := 1, Execute := TRUE);
			IF fb_RunLayerPad.Complete THEN
				fb_RunLayerPad(Execute := FALSE);
				FG_sequence := 6;
			ELSIF fb_RunLayerPad.Error THEN
				fb_RunLayerPad(Execute := FALSE);
				AUTO_MODE.Halt_Production := TRUE;
				FG_sequence := 6;
			END_IF
		ELSIF GVL.Basket_A_Counter = 30 THEN
			fb_RunLayerPad(Basket := 1, Layer := 2, Execute := TRUE);
			IF fb_RunLayerPad.Complete THEN
				fb_RunLayerPad(Execute := FALSE);
				FG_sequence := 6;
			ELSIF fb_RunLayerPad.Error THEN
				fb_RunLayerPad(Execute := FALSE);
				AUTO_MODE.Halt_Production := TRUE;
				FG_sequence := 6;
			END_IF
		ELSIF GVL.Basket_A_Counter = 45 THEN
			fb_RunLayerPad(Basket := 1, Layer := 3, Execute := TRUE);
			IF fb_RunLayerPad.Complete THEN
				fb_RunLayerPad(Execute := FALSE);
				FG_sequence := 6;
			ELSIF fb_RunLayerPad.Error THEN
				fb_RunLayerPad(Execute := FALSE);
				AUTO_MODE.Halt_Production := TRUE;
				FG_sequence := 6;
			END_IF
		ELSIF GVL.Basket_A_Counter = 60 THEN
			fb_RunLayerPad(Basket := 1, Layer := 4, Execute := TRUE);
			IF fb_RunLayerPad.Complete THEN
				fb_RunLayerPad(Execute := FALSE);
				FG_sequence := 6;
			ELSIF fb_RunLayerPad.Error THEN
				fb_RunLayerPad(Execute := FALSE);
				AUTO_MODE.Halt_Production := TRUE;
				FG_sequence := 6;
			END_IF
		ELSIF GVL.Basket_A_Counter = 75 THEN
			fb_RunLayerPad(Basket := 1, Layer := 5, Execute := TRUE);
			IF fb_RunLayerPad.Complete THEN
				fb_RunLayerPad(Execute := FALSE);
				FG_sequence := 6;
			ELSIF fb_RunLayerPad.Error THEN
				fb_RunLayerPad(Execute := FALSE);
				AUTO_MODE.Halt_Production := TRUE;
				FG_sequence := 6;
			END_IF
		ELSIF GVL.Basket_A_Counter = 90 THEN
			fb_RunLayerPad(Basket := 1, Layer := 6, Execute := TRUE);
			IF fb_RunLayerPad.Complete THEN
				fb_RunLayerPad(Execute := FALSE);
				FG_sequence := 6;
			ELSIF fb_RunLayerPad.Error THEN
				fb_RunLayerPad(Execute := FALSE);
				AUTO_MODE.Halt_Production := TRUE;
				FG_sequence := 6;
			END_IF
		ELSIF GVL.Basket_A_Counter = 100 THEN
			fb_RunLayerPad(Basket := 1, Layer := 7, Execute := TRUE);
			IF fb_RunLayerPad.Complete THEN
				fb_RunLayerPad(Execute := FALSE);
				FG_sequence := 6;
			ELSIF fb_RunLayerPad.Error THEN
				fb_RunLayerPad(Execute := FALSE);
				AUTO_MODE.Halt_Production := TRUE;
			END_IF
		ELSE
			FG_sequence := 6;
		END_IF
		
	6:
		FG_sequence := 0;
		AUTO_MODE.next_step := FALSE;
		AUTO_MODE.FG_PACKING := FALSE;
		AUTO_MODE.processnameFG := CONCAT(MSG.COMP_FG,MAIN.fb_TimeStamp.SystemTime);
		AUTO_MODE.processnameFG := CONCAT(AUTO_MODE.processnameFG,MSG.STATUS_END);
		LOGPROCESS( spLogComp	 := MSG.COMP_FG, 
					spLogAction	 := MSG.ACTION_FG_PACK, 
					spLogStatus	 := MSG.STATUS_END,
					plogFlag	 := TRUE);
END_CASE

END_PROGRAM

// ---- POUs/Auto_Seq/FB_RunLayerPad.TcPOU
FUNCTION_BLOCK FB_RunLayerPad
VAR
	LP_sequence	: UINT;
	
	process_A	: UINT; //KR5 Remove Magnet
	process_B	: UINT; //KR5 Get Suction
	process_C	: UINT; //KR5 Get Layer Pad
	process_D	: UINT; //KR5 Place Layer Pad
	process_E	: UINT; //KR5 Remove Suction
	process_F	: UINT; //KR5 Get Magnet
	
	bit1		: UINT;
	bit2		: UINT;
	
END_VAR
VAR_INPUT
	Basket 		: UINT;
	Layer		: UINT;
	Execute		: BOOL;
END_VAR
VAR_OUTPUT
	Complete	: BOOL;
	Error		: BOOL;
END_VAR

IF NOT Execute THEN
	 LP_sequence := 0;
	 RETURN;	
END_IF

CASE LP_sequence OF
	// Init ------------------------------------------------------------------------------------------------------------------	
	0:
		AUTO_MODE.processnameFG := CONCAT(MSG.COMP_FG,MSG.ACTION_LYRPD_INIT);	
		LOGPROCESS( spLogComp	 := MSG.COMP_FG, 
		 			spLogAction	 := MSG.ACTION_LYRPD_INIT, 
		 			spLogStatus	 := MSG.STATUS_DONE,
	 	 		 	plogFlag	 := TRUE);
		process_A	:= 0;
		process_B	:= 0;
		process_C	:= 0;
		process_D	:= 0;
		process_E	:= 0;
		Error 		:= FALSE;
		Complete	:= FALSE;
		LP_sequence := 1;
		GVL.LAYERPAD := TRUE;
	
	// Check Tool -------------------------------------------------------------------------------------------------------------	
	1:	
		IF GVL.KR1_EOAT_FILL THEN
			// Remove Magnet EOAT
			IF process_A = 0 THEN
				IF KR1.Idle THEN
//					KR1.PLC_O_D3.1 := TRUE; //201
					KR1.bOutBit[3,1] := TRUE;
					AUTO_MODE.processnameFG := CONCAT(MSG.COMP_FG,MSG.ACTION_REMOVE_MAGNET);
					AUTO_MODE.processnameFG := CONCAT(AUTO_MODE.processnameFG,MSG.STATUS_RUN);
					LOGPROCESS( spLogComp	 := MSG.COMP_FG, 
								spLogAction	 := MSG.ACTION_REMOVE_MAGNET, 
								spLogStatus	 := MSG.STATUS_RUN,
								plogFlag	 := TRUE);
					process_A := 1;
					RETURN;
				END_IF
			ELSIF process_A = 1 THEN
//				KR1.PLC_O_D3.1 := TRUE; //201
				KR1.bOutBit[3,1] := TRUE;
				IF KR1.bInBit[3,1] THEN
//					KR1.PLC_O_D3.1 := FALSE; //201
					KR1.bOutBit[3,1] := FALSE;
					AUTO_MODE.processnameFG := CONCAT(MSG.COMP_FG,MSG.ACTION_REMOVE_MAGNET);
					AUTO_MODE.processnameFG := CONCAT(AUTO_MODE.processnameFG,MSG.STATUS_ACK);
					LOGPROCESS( spLogComp	 := MSG.COMP_FG, 
								spLogAction	 := MSG.ACTION_REMOVE_MAGNET, 
								spLogStatus	 := MSG.STATUS_ACK,
								plogFlag	 := TRUE);
					process_A := 2;
					RETURN;
				END_IF	
			ELSIF process_A = 2 THEN
//				KR1.PLC_O_D3.1 := FALSE; //201
				KR1.bOutBit[3,1] := FALSE;
				IF NOT KR1.bInBit[3,1] THEN
					AUTO_MODE.processnameFG := CONCAT(MSG.COMP_FG,MSG.ACTION_REMOVE_MAGNET);
					AUTO_MODE.processnameFG := CONCAT(AUTO_MODE.processnameFG,MSG.STATUS_DONE);
					LOGPROCESS( spLogComp	 := MSG.COMP_FG, 
								spLogAction	 := MSG.ACTION_REMOVE_MAGNET, 
								spLogStatus	 := MSG.STATUS_DONE,
								plogFlag	 := TRUE);
					process_A:= 3;
					RETURN;
				END_IF	
			ELSIF process_A = 3 THEN
				IF KR1.Idle THEN
					AUTO_MODE.processnameFG := CONCAT(MSG.COMP_FG,MSG.ACTION_REMOVE_MAGNET);
					AUTO_MODE.processnameFG := CONCAT(AUTO_MODE.processnameFG,MSG.STATUS_COMP);
					LOGPROCESS( spLogComp	 := MSG.COMP_FG, 
								spLogAction	 := MSG.ACTION_REMOVE_MAGNET, 
								spLogStatus	 := MSG.STATUS_COMP,
								plogFlag	 := TRUE);
					process_A := 4;
					LP_sequence := 2;
					AUTO_MODE.next_step := FALSE;
					GVL.KR1_EOAT_FILL := FALSE;
				END_IF
			END_IF
		ELSE
			LP_sequence := 2;
		END_IF
	
	// Get Suction -------------------------------------------------------------------------------------------------------------	
	2:	
		IF NOT GVL.KR1_EOAT_FILL AND NOT GVL.KR1_EOAT_SUCTION THEN
			// Get Suction EOAT
			IF process_B = 0 THEN
				IF KR1.Idle THEN
//					KR1.PLC_O_D3.2 := TRUE; //202
					KR1.bOutBit[3,2] := TRUE;
					AUTO_MODE.processnameFG := CONCAT(MSG.COMP_FG,MSG.ACTION_GET_SUCTION);
					AUTO_MODE.processnameFG := CONCAT(AUTO_MODE.processnameFG,MSG.STATUS_RUN);
					LOGPROCESS( spLogComp	 := MSG.COMP_FG, 
								spLogAction	 := MSG.ACTION_GET_SUCTION, 
								spLogStatus	 := MSG.STATUS_RUN,
								plogFlag	 := TRUE);
					process_B := 1;
					RETURN;
				END_IF
			ELSIF process_B = 1 THEN
//				KR1.PLC_O_D3.2 := TRUE; //202
				KR1.bOutBit[3,2] := TRUE;
				IF KR1.bInBit[3,2] THEN
//					KR1.PLC_O_D3.2 := FALSE; //202	
					KR1.bOutBit[3,2] := FALSE;
					AUTO_MODE.processnameFG := CONCAT(MSG.COMP_FG,MSG.ACTION_GET_SUCTION);
					AUTO_MODE.processnameFG := CONCAT(AUTO_MODE.processnameFG,MSG.STATUS_ACK);
					LOGPROCESS( spLogComp	 := MSG.COMP_FG, 
								spLogAction	 := MSG.ACTION_GET_SUCTION, 
								spLogStatus	 := MSG.STATUS_ACK,
								plogFlag	 := TRUE);
					process_B := 2;
					RETURN;
				END_IF	
			ELSIF process_B = 2 THEN
//				KR1.PLC_O_D3.2 := FALSE; //202	
				KR1.bOutBit[3,2] := FALSE;
				IF NOT KR1.bInBit[3,2] THEN
					AUTO_MODE.processnameFG := CONCAT(MSG.COMP_FG,MSG.ACTION_GET_SUCTION);
					AUTO_MODE.processnameFG := CONCAT(AUTO_MODE.processnameFG,MSG.STATUS_DONE);
					LOGPROCESS( spLogComp	 := MSG.COMP_FG, 
								spLogAction	 := MSG.ACTION_GET_SUCTION, 
								spLogStatus	 := MSG.STATUS_DONE,
								plogFlag	 := TRUE);
					process_B:= 3;
					RETURN;
				END_IF	
			ELSIF process_B = 3 THEN
				IF KR1.Idle THEN
					AUTO_MODE.processnameFG := CONCAT(MSG.COMP_FG,MSG.ACTION_GET_SUCTION);
					AUTO_MODE.processnameFG := CONCAT(AUTO_MODE.processnameFG,MSG.STATUS_COMP);
					LOGPROCESS( spLogComp	 := MSG.COMP_FG, 
								spLogAction	 := MSG.ACTION_GET_SUCTION, 
								spLogStatus	 := MSG.STATUS_COMP,
								plogFlag	 := TRUE);
					process_B := 4;
					LP_sequence := 4;
					AUTO_MODE.next_step := FALSE;
					GVL.KR1_EOAT_SUCTION := TRUE;
				END_IF
			END_IF
		ELSE
			LP_sequence := 4;
		END_IF
	
	// Get Layer Pad -------------------------------------------------------------------------------------------------------------	
//	3:	
//		IF GVL.KR1_EOAT_SUCTION THEN
//			// Get Layer Pad
//			IF process_C = 0 THEN
//				IF KR1.Idle THEN
//					KR1.PLC_O_D4.1 := TRUE; //202
//					AUTO_MODE.processnameFG := CONCAT(MSG.COMP_FG,MSG.ACTION_GET_LAYER_PAD);
//					AUTO_MODE.processnameFG := CONCAT(AUTO_MODE.processnameFG,MSG.STATUS_RUN);
//					LOGPROCESS( spLogComp	 := MSG.COMP_FG, 
//								spLogAction	 := MSG.ACTION_GET_LAYER_PAD, 
//								spLogStatus	 := MSG.STATUS_RUN,
//								plogFlag	 := TRUE);
//					process_C := 1;
//					RETURN;
//				END_IF
//			ELSIF process_C = 1 THEN
//				KR1.PLC_O_D4.1 := TRUE; //202
//				IF KR1.bInBit[4,1] THEN
//					KR1.PLC_O_D4.1 := FALSE; //202	
//					AUTO_MODE.processnameFG := CONCAT(MSG.COMP_FG,MSG.ACTION_GET_LAYER_PAD);
//					AUTO_MODE.processnameFG := CONCAT(AUTO_MODE.processnameFG,MSG.STATUS_ACK);
//					LOGPROCESS( spLogComp	 := MSG.COMP_FG, 
//								spLogAction	 := MSG.ACTION_GET_LAYER_PAD, 
//								spLogStatus	 := MSG.STATUS_ACK,
//								plogFlag	 := TRUE);
//					process_C := 2;
//					RETURN;
//				END_IF	
//			ELSIF process_C = 2 THEN
//				KR1.PLC_O_D4.1 := FALSE; //202	
//				IF NOT KR1.bInBit[4,1] THEN
//					AUTO_MODE.processnameFG := CONCAT(MSG.COMP_FG,MSG.ACTION_GET_LAYER_PAD);
//					AUTO_MODE.processnameFG := CONCAT(AUTO_MODE.processnameFG,MSG.STATUS_DONE);
//					LOGPROCESS( spLogComp	 := MSG.COMP_FG, 
//								spLogAction	 := MSG.ACTION_GET_LAYER_PAD, 
//								spLogStatus	 := MSG.STATUS_DONE,
//								plogFlag	 := TRUE);
//					process_C:= 3;
//					RETURN;
//				END_IF	
//			ELSIF process_C = 3 THEN
//				IF KR1.Idle THEN
//					AUTO_MODE.processnameFG := CONCAT(MSG.COMP_FG,MSG.ACTION_GET_LAYER_PAD);
//					AUTO_MODE.processnameFG := CONCAT(AUTO_MODE.processnameFG,MSG.STATUS_COMP);
//					LOGPROCESS( spLogComp	 := MSG.COMP_FG, 
//								spLogAction	 := MSG.ACTION_GET_LAYER_PAD, 
//								spLogStatus	 := MSG.STATUS_COMP,
//								plogFlag	 := TRUE);
//					process_C := 4;
//					LP_sequence := 4;
//					AUTO_MODE.next_step := FALSE;
//					GVL.KR1_EOAT_SUCTION := TRUE;
//				END_IF
//			END_IF
//		ELSE
//			Error := TRUE;
//		END_IF
		
	// Place Layer Pad -------------------------------------------------------------------------------------------------------------	
	4:	
		IF Basket = 1 THEN
			CASE Layer OF
				0:
					bit1 := 29;
					bit2 := 2;
				1:
					bit1 := 29;
					bit2 := 3;
				2:
					bit1 := 29;
					bit2 := 4;
				3:
					bit1 := 29;
					bit2 := 5;
				4:
					bit1 := 29;
					bit2 := 6;
				5:
					bit1 := 29;
					bit2 := 7;
				6:
					bit1 := 30;
					bit2 := 0;
				7:
					bit1 := 30;
					bit2 := 1;
				8:
					bit1 := 30;
					bit2 := 2;
				9:
					bit1 := 30;
					bit2 := 3;
			END_CASE	
		END_IF
		
		IF GVL.KR1_EOAT_SUCTION THEN
			// Place Layer Pad
			IF process_D = 0 THEN
				IF KR1.Idle THEN
					KR1.bOutBit[bit1,bit2] := TRUE;
//					KR1.PLC_O_D4.1 := TRUE; //202
					AUTO_MODE.processnameFG := CONCAT(MSG.COMP_FG,MSG.ACTION_PLACE_LAYER_PAD);
					AUTO_MODE.processnameFG := CONCAT(AUTO_MODE.processnameFG,MSG.STATUS_RUN);
					LOGPROCESS( spLogComp	 := MSG.COMP_FG, 
								spLogAction	 := MSG.ACTION_PLACE_LAYER_PAD, 
								spLogStatus	 := MSG.STATUS_RUN,
								plogFlag	 := TRUE);
					process_D := 1;
					RETURN;
				END_IF
			ELSIF process_D = 1 THEN
				KR1.bOutBit[bit1,bit2] := TRUE;
//				KR1.PLC_O_D4.1 := TRUE; //202
				IF KR1.bInBit[bit1,bit2] THEN
					KR1.bOutBit[bit1,bit2] := FALSE;
//					KR1.PLC_O_D4.1 := FALSE; //202	
					AUTO_MODE.processnameFG := CONCAT(MSG.COMP_FG,MSG.ACTION_PLACE_LAYER_PAD);
					AUTO_MODE.processnameFG := CONCAT(AUTO_MODE.processnameFG,MSG.STATUS_ACK);
					LOGPROCESS( spLogComp	 := MSG.COMP_FG, 
								spLogAction	 := MSG.ACTION_PLACE_LAYER_PAD, 
								spLogStatus	 := MSG.STATUS_ACK,
								plogFlag	 := TRUE);
					process_D := 2;
					RETURN;
				END_IF	
			ELSIF process_D = 2 THEN
				KR1.bOutBit[bit1,bit2] := FALSE;
//				KR1.PLC_O_D4.1 := FALSE; //202	
				IF NOT KR1.bInBit[bit1,bit2] THEN
					AUTO_MODE.processnameFG := CONCAT(MSG.COMP_FG,MSG.ACTION_PLACE_LAYER_PAD);
					AUTO_MODE.processnameFG := CONCAT(AUTO_MODE.processnameFG,MSG.STATUS_DONE);
					LOGPROCESS( spLogComp	 := MSG.COMP_FG, 
								spLogAction	 := MSG.ACTION_PLACE_LAYER_PAD, 
								spLogStatus	 := MSG.STATUS_DONE,
								plogFlag	 := TRUE);
					process_D:= 3;
					RETURN;
				END_IF	
			ELSIF process_D = 3 THEN
				IF KR1.Idle THEN
					AUTO_MODE.processnameFG := CONCAT(MSG.COMP_FG,MSG.ACTION_PLACE_LAYER_PAD);
					AUTO_MODE.processnameFG := CONCAT(AUTO_MODE.processnameFG,MSG.STATUS_COMP);
					LOGPROCESS( spLogComp	 := MSG.COMP_FG, 
								spLogAction	 := MSG.ACTION_PLACE_LAYER_PAD, 
								spLogStatus	 := MSG.STATUS_COMP,
								plogFlag	 := TRUE);
					process_D := 4;
					LP_sequence := 5;
					AUTO_MODE.next_step := FALSE;
					GVL.KR1_EOAT_SUCTION := TRUE;
				END_IF
			END_IF
		ELSE
			Error := TRUE;
		END_IF
		
	// Remove Suction -------------------------------------------------------------------------------------------------------------	
	5:	
		IF GVL.KR1_EOAT_SUCTION THEN
			// Remove Layer Pad
			IF process_E = 0 THEN
				IF KR1.Idle THEN
//					KR1.PLC_O_D3.3 := TRUE; //203
					KR1.bOutBit[3,3] := TRUE;
					AUTO_MODE.processnameFG := CONCAT(MSG.COMP_FG,MSG.ACTION_REMOVE_SUCTION);
					AUTO_MODE.processnameFG := CONCAT(AUTO_MODE.processnameFG,MSG.STATUS_RUN);
					LOGPROCESS( spLogComp	 := MSG.COMP_FG, 
								spLogAction	 := MSG.ACTION_REMOVE_SUCTION, 
								spLogStatus	 := MSG.STATUS_RUN,
								plogFlag	 := TRUE);
					process_E := 1;
					RETURN;
				END_IF
			ELSIF process_E = 1 THEN
//				KR1.PLC_O_D3.3 := TRUE; //203
				KR1.bOutBit[3,3] := TRUE;
				IF KR1.bInBit[3,3] THEN
//					KR1.PLC_O_D3.3 := FALSE; //203	
					KR1.bOutBit[3,3] := FALSE;
					AUTO_MODE.processnameFG := CONCAT(MSG.COMP_FG,MSG.ACTION_REMOVE_SUCTION);
					AUTO_MODE.processnameFG := CONCAT(AUTO_MODE.processnameFG,MSG.STATUS_ACK);
					LOGPROCESS( spLogComp	 := MSG.COMP_FG, 
								spLogAction	 := MSG.ACTION_REMOVE_SUCTION, 
								spLogStatus	 := MSG.STATUS_ACK,
								plogFlag	 := TRUE);
					process_E := 2;
					RETURN;
				END_IF	
			ELSIF process_E = 2 THEN
//				KR1.PLC_O_D3.3 := FALSE; //203	
				KR1.bOutBit[3,3] := FALSE;
				IF NOT KR1.bInBit[3,3] THEN
					AUTO_MODE.processnameFG := CONCAT(MSG.COMP_FG,MSG.ACTION_REMOVE_SUCTION);
					AUTO_MODE.processnameFG := CONCAT(AUTO_MODE.processnameFG,MSG.STATUS_DONE);
					LOGPROCESS( spLogComp	 := MSG.COMP_FG, 
								spLogAction	 := MSG.ACTION_REMOVE_SUCTION, 
								spLogStatus	 := MSG.STATUS_DONE,
								plogFlag	 := TRUE);
					process_E:= 3;
					RETURN;
				END_IF	
			ELSIF process_E = 3 THEN
				IF KR1.Idle THEN
					AUTO_MODE.processnameFG := CONCAT(MSG.COMP_FG,MSG.ACTION_REMOVE_SUCTION);
					AUTO_MODE.processnameFG := CONCAT(AUTO_MODE.processnameFG,MSG.STATUS_COMP);
					LOGPROCESS( spLogComp	 := MSG.COMP_FG, 
								spLogAction	 := MSG.ACTION_REMOVE_SUCTION, 
								spLogStatus	 := MSG.STATUS_COMP,
								plogFlag	 := TRUE);
					process_E := 4;
					LP_sequence := 6;
					AUTO_MODE.next_step := FALSE;
					GVL.KR1_EOAT_SUCTION := FALSE;
				END_IF
			END_IF
		ELSE
			Error := TRUE;
		END_IF
		
	// Get Magnet --------------------------------------------------------------------------------------------------------------	
	6:	
		IF NOT GVL.KR1_EOAT_FILL AND NOT GVL.KR1_EOAT_SUCTION THEN
			IF process_F = 0 THEN
				IF KR1.Idle THEN
//					KR1.PLC_O_D3.0 := TRUE; //200
					KR1.bOutBit[3,0] := TRUE;
								AUTO_MODE.processnameFG := CONCAT(MSG.COMP_FG,MSG.ACTION_GET_MAGNET);
								AUTO_MODE.processnameFG := CONCAT(AUTO_MODE.processnameFG,MSG.STATUS_RUN);
								LOGPROCESS( spLogComp	 := MSG.COMP_FG, 
											spLogAction	 := MSG.ACTION_GET_MAGNET, 
											spLogStatus	 := MSG.STATUS_RUN,
											plogFlag	 := TRUE);
					process_F := 1;
					RETURN;
				END_IF
			ELSIF process_F = 1 THEN
//				KR1.PLC_O_D3.0 := TRUE; //200
				KR1.bOutBit[3,0] := TRUE;
				IF NOT KR1.bInBit[3,0] THEN
//					KR1.PLC_O_D3.0 := FALSE; //200	
					KR1.bOutBit[3,0] := FALSE;
					AUTO_MODE.processnameFG := CONCAT(MSG.COMP_FG,MSG.ACTION_GET_MAGNET);
					AUTO_MODE.processnameFG := CONCAT(AUTO_MODE.processnameFG,MSG.STATUS_ACK);
					LOGPROCESS( spLogComp	 := MSG.COMP_FG, 
								spLogAction	 := MSG.ACTION_GET_MAGNET, 
								spLogStatus	 := MSG.STATUS_ACK,
								plogFlag	 := TRUE);
					process_F := 2;
					RETURN;
				END_IF	
			ELSIF process_F = 2 THEN
//				KR1.PLC_O_D3.0 := FALSE; //200	
				KR1.bOutBit[3,0] := FALSE;
				IF KR1.bInBit[3,0] THEN
					AUTO_MODE.processnameFG := CONCAT(MSG.COMP_FG,MSG.ACTION_GET_MAGNET);
					AUTO_MODE.processnameFG := CONCAT(AUTO_MODE.processnameFG,MSG.STATUS_DONE);
					LOGPROCESS( spLogComp	 := MSG.COMP_FG, 
								spLogAction	 := MSG.ACTION_GET_MAGNET, 
								spLogStatus	 := MSG.STATUS_DONE,
								plogFlag	 := TRUE);
					process_F:= 3;
					RETURN;
				END_IF	
			ELSIF process_F = 3 THEN
				IF KR1.Idle THEN
					AUTO_MODE.processnameFG := CONCAT(MSG.COMP_FG,MSG.ACTION_GET_MAGNET);
					AUTO_MODE.processnameFG := CONCAT(AUTO_MODE.processnameFG,MSG.STATUS_COMP);
					LOGPROCESS( spLogComp	 := MSG.COMP_FG, 
								spLogAction	 := MSG.ACTION_GET_MAGNET, 
								spLogStatus	 := MSG.STATUS_COMP,
								plogFlag	 := TRUE);
					process_F := 4;
					LP_sequence := 7;
					AUTO_MODE.next_step := FALSE;
					GVL.KR1_EOAT_FILL := TRUE;
				END_IF
			END_IF
		ELSE
			Error := TRUE;
		END_IF
		
	// Complete ---------------------------------------------------------------------------------------------------------------	
	7:
		GVL.LAYERPAD := FALSE;
		Complete := TRUE;	
		
END_CASE

END_FUNCTION_BLOCK

// ---- POUs/Auto_Seq/SEQ_COSMO.TcPOU
PROGRAM SEQ_COSMO
VAR_INPUT
	COSMO_sequence	: UINT;
END_VAR

VAR
	process_V	: UINT; //COSMO to Pitstop
	process_W	: UINT; //COSMO to Reject Out
	process_X	: UINT; //Conveyor to Pitstop
	process_G	: UINT; //KR1 GET Magnet	
END_VAR


IF NOT AUTO_MODE.COSMO_LOAD OR GVL.KR1_EOAT_SUCTION OR GVL.LAYERPAD OR AUTO_MODE.FG_PACKING THEN
	RETURN;
END_IF

CASE COSMO_sequence OF
	0:
		process_V	:= 0;
		process_W	:= 0;
		process_X	:= 0;
		process_G	:= 0;
		COSMO_sequence := 1;		
		GVL.COSMO_UNLOAD := TRUE;
		AUTO_MODE.processnameCOSMO := CONCAT(MSG.COMP_CM,MSG.ACTION_INIT);
		LOGPROCESS( spLogComp	 := MSG.COMP_CM, 
		 			spLogAction	 := MSG.ACTION_INIT, 
		 			spLogStatus	 := MSG.STATUS_DONE,
	 	 		 	plogFlag	 := TRUE);
		
	// Get Magnet -------------------------------------------------------------------------------------------------------------	
	1:
		IF NOT GVL.KR1_EOAT_FILL AND NOT GVL.KR1_EOAT_SUCTION THEN
			IF process_G = 0 THEN
				IF KR1.Idle THEN
//					KR1.PLC_O_D3.0 := TRUE; //200
					KR1.bOutBit[3,0] := TRUE;
					AUTO_MODE.processnameCOSMO := CONCAT(MSG.COMP_CM,MSG.ACTION_GET_MAGNET);
					AUTO_MODE.processnameCOSMO := CONCAT(AUTO_MODE.processnameCOSMO,MSG.STATUS_RUN);
					LOGPROCESS( spLogComp	 := MSG.COMP_CM, 
								spLogAction	 := MSG.ACTION_GET_MAGNET, 
								spLogStatus	 := MSG.STATUS_RUN,
								plogFlag	 := TRUE);
					process_G := 1;
					RETURN;
				END_IF
			ELSIF process_G = 1 THEN
//				KR1.PLC_O_D3.0 := TRUE; //200
				KR1.bOutBit[3,0] := TRUE;
				IF NOT KR1.bInBit[3,0] THEN
//					KR1.PLC_O_D3.0 := FALSE; //200	
					KR1.bOutBit[3,0] := FALSE;
					AUTO_MODE.processnameCOSMO := CONCAT(MSG.COMP_CM,MSG.ACTION_GET_MAGNET);
					AUTO_MODE.processnameCOSMO := CONCAT(AUTO_MODE.processnameCOSMO,MSG.STATUS_ACK);
					LOGPROCESS( spLogComp	 := MSG.COMP_CM, 
								spLogAction	 := MSG.ACTION_GET_MAGNET, 
								spLogStatus	 := MSG.STATUS_ACK,
								plogFlag	 := TRUE);
					process_G := 2;
					RETURN;
				END_IF	
			ELSIF process_G = 2 THEN
//				KR1.PLC_O_D3.0 := FALSE; //200
				KR1.bOutBit[3,0] := FALSE;	
				IF KR1.bInBit[3,0] THEN
					AUTO_MODE.processnameCOSMO := CONCAT(MSG.COMP_CM,MSG.ACTION_GET_MAGNET);
					AUTO_MODE.processnameCOSMO := CONCAT(AUTO_MODE.processnameCOSMO,MSG.STATUS_DONE);
					LOGPROCESS( spLogComp	 := MSG.COMP_CM, 
								spLogAction	 := MSG.ACTION_GET_MAGNET, 
								spLogStatus	 := MSG.STATUS_DONE,
								plogFlag	 := TRUE);
					process_G:= 3;
					RETURN;
				END_IF	
			ELSIF process_G = 3 THEN
				IF KR1.Idle THEN
					AUTO_MODE.processnameCOSMO := CONCAT(MSG.COMP_CM,MSG.ACTION_GET_MAGNET);
					AUTO_MODE.processnameCOSMO := CONCAT(AUTO_MODE.processnameCOSMO,MSG.STATUS_COMP);
					LOGPROCESS( spLogComp	 := MSG.COMP_CM, 
								spLogAction	 := MSG.ACTION_GET_MAGNET, 
								spLogStatus	 := MSG.STATUS_COMP,
								plogFlag	 := TRUE);
					process_G := 4;
					COSMO_sequence := 2;
					AUTO_MODE.next_step := FALSE;
					GVL.KR1_EOAT_FILL := TRUE;
				END_IF
			END_IF
		ELSE
			COSMO_sequence := 2;
		END_IF
		
	// COSMO test --------------------------------------------------------------------------------------------------------------		
	2: 
		IF GVL.COSMO_OK THEN
			GVL.COSMO_Run := FALSE;
			AUTO_MODE.COSMO_RUN := FALSE;
			AUTO_MODE.processnameCOSMO := CONCAT(MSG.COMP_CM,MSG.ACTION_COSMO_PASS);
			AUTO_MODE.processnameCOSMO := CONCAT(AUTO_MODE.processnameCOSMO,MSG.STATUS_DONE);
			LOGPROCESS( spLogComp	 := MSG.COMP_CM, 
						spLogAction	 := MSG.ACTION_COSMO_PASS, 
						spLogStatus	 := MSG.STATUS_DONE,
						plogFlag	 := TRUE);
			COSMO_sequence := 3;
			AUTO_MODE.next_step := FALSE;
			AUTO_MODE.CLEAR_COSMO := TRUE;
			RETURN;
		ELSIF GVL.COSMO_NOTOK THEN
			GVL.COSMO_Run := FALSE;
			AUTO_MODE.COSMO_RUN := FALSE;
			AUTO_MODE.processnameCOSMO := CONCAT(MSG.COMP_CM,MSG.ACTION_COSMO_FAIL);
			AUTO_MODE.processnameCOSMO := CONCAT(AUTO_MODE.processnameCOSMO,MSG.STATUS_DONE);
			LOGPROCESS( spLogComp	 := MSG.COMP_CM, 
						spLogAction	 := MSG.ACTION_COSMO_FAIL, 
						spLogStatus	 := MSG.STATUS_DONE,
						plogFlag	 := TRUE);
			COSMO_sequence := 3;
			AUTO_MODE.next_step := FALSE;
			AUTO_MODE.CLEAR_COSMO := TRUE;
			RETURN;
		END_IF
			
	// COSMO to Reject Out -------------------------------------------------------------------------------------------------------------	
	3: 
			IF process_W = 0 THEN
				IF NOT AUTO_MODE.KR1_PITSTOP AND KR1.Idle AND NOT GVL.Conveyor_Full AND GVL.KR1_EOAT_FILL AND NOT AUTO_MODE.FG_PACKING AND NOT AUTO_MODE.RW_PACKING THEN
					KR1.bOutBit[3,6] := TRUE; //206
					AUTO_MODE.processnameCOSMO := CONCAT(MSG.COMP_CM,MSG.ACTION_COSMO_TO_CNVYR);
					AUTO_MODE.processnameCOSMO := CONCAT(AUTO_MODE.processnameCOSMO,MSG.STATUS_RUN);
					LOGPROCESS( spLogComp	 := MSG.COMP_CM, 
								spLogAction	 := MSG.ACTION_COSMO_TO_CNVYR, 
								spLogStatus	 := MSG.STATUS_RUN,
								plogFlag	 := TRUE);
					process_W := 1;
					RETURN;
				END_IF
			ELSIF process_W = 1 THEN
				KR1.bOutBit[3,6]:= TRUE; //206
				IF KR1.bInBit[3,6] THEN
					KR1.bOutBit[3,6] := FALSE; //2056
					AUTO_MODE.processnameCOSMO := CONCAT(MSG.COMP_CM,MSG.ACTION_COSMO_TO_CNVYR);
					AUTO_MODE.processnameCOSMO := CONCAT(AUTO_MODE.processnameCOSMO,MSG.STATUS_ACK);
					LOGPROCESS( spLogComp	 := MSG.COMP_CM, 
								spLogAction	 := MSG.ACTION_COSMO_TO_CNVYR, 
								spLogStatus	 := MSG.STATUS_ACK,
								plogFlag	 := TRUE);
					process_W := 2;
					RETURN;
				END_IF	
			ELSIF process_W = 2 THEN
				KR1.bOutBit[3,6] := FALSE; //206
				IF NOT KR1.bInBit[3,6] THEN
					AUTO_MODE.processnameCOSMO := CONCAT(MSG.COMP_CM,MSG.ACTION_COSMO_TO_CNVYR);
					AUTO_MODE.processnameCOSMO := CONCAT(AUTO_MODE.processnameCOSMO,MSG.STATUS_DONE);
					LOGPROCESS( spLogComp	 := MSG.COMP_CM, 
								spLogAction	 := MSG.ACTION_COSMO_TO_CNVYR, 
								spLogStatus	 := MSG.STATUS_DONE,
								plogFlag	 := TRUE);
					process_W:= 3;
					RETURN;
				END_IF
			ELSIF process_W = 3 THEN
				IF KR1.Idle THEN
						AUTO_MODE.processnameCOSMO := CONCAT(MSG.COMP_CM,MSG.ACTION_COSMO_TO_CNVYR);
						AUTO_MODE.processnameCOSMO := CONCAT(AUTO_MODE.processnameCOSMO,MSG.STATUS_COMP);
						LOGPROCESS( spLogComp	 := MSG.COMP_CM, 
									spLogAction	 := MSG.ACTION_COSMO_TO_CNVYR, 
									spLogStatus	 := MSG.STATUS_COMP,
									plogFlag	 := TRUE);
						process_W := 4;
						COSMO_sequence := 4;
						AUTO_MODE.next_step := FALSE;
						AUTO_MODE.CR_UNLOADING := FALSE;
						AUTO_MODE.CLEAR_COSMO := FALSE;
						GVL.Fail_Counter := GVL.Fail_Counter+1;
					END_IF
			END_IF	
	
	4:
		COSMO_sequence := 0;
		AUTO_MODE.next_step := FALSE;
		AUTO_MODE.COSMO_LOAD := FALSE;
		AUTO_MODE.CR_UNLOADING := FALSE;
		AUTO_MODE.CLEAR_COSMO := FALSE;
		GVL.COSMO_UNLOAD := FALSE;
		AUTO_MODE.processnameCOSMO := CONCAT(MSG.COMP_CM,MAIN.fb_TimeStamp.SystemTime);
		AUTO_MODE.processnameCOSMO := CONCAT(AUTO_MODE.processnameCOSMO,MSG.STATUS_END);
		AUTO_MODE.processnameCOSMO := CONCAT(MSG.COMP_CM,MSG.ACTION_COSMO);
		AUTO_MODE.processnameCOSMO := CONCAT(AUTO_MODE.processnameCOSMO,MSG.STATUS_END);
		LOGPROCESS( spLogComp	 := MSG.COMP_CM, 
					spLogAction	 := MSG.ACTION_COSMO, 
					spLogStatus	 := MSG.STATUS_END,
					plogFlag	 := TRUE);
END_CASE

END_PROGRAM

// ---- POUs/Auto_Seq/SEQ_RW.TcPOU
PROGRAM SEQ_RW
VAR_INPUT
	RW_sequence	: UINT;
END_VAR

VAR
	process_X	: UINT; //Conveyor to Pitstop
	process_G	: UINT; //KR1 GET Magnet	
END_VAR


IF AUTO_MODE.KR1_PITSTOP THEN
	RETURN;
END_IF

CASE RW_sequence OF
	0:
		AUTO_MODE.processnameCR := CONCAT(MSG.COMP_RW,MSG.ACTION_INIT);	
		LOGPROCESS( spLogComp	 := MSG.COMP_RW, 
		 			spLogAction	 := MSG.ACTION_INIT, 
		 			spLogStatus	 := MSG.STATUS_DONE,
	 	 		 	plogFlag	 := TRUE);
		process_X	:= 0;
		process_G	:= 0;
		RW_sequence := 1;
		
	// Get Magnet -------------------------------------------------------------------------------------------------------------	
	1:
		IF NOT GVL.KR1_EOAT_FILL THEN
			IF process_G = 0 THEN
				IF KR1.Idle THEN
//					KR1.PLC_O_D3.0 := TRUE; //200
					KR1.bOutBit[3,0] := TRUE;
					AUTO_MODE.processnameCOSMO := CONCAT(MSG.COMP_RW,MSG.ACTION_GET_MAGNET);
					AUTO_MODE.processnameCOSMO := CONCAT(AUTO_MODE.processnameCOSMO,MSG.STATUS_RUN);
					LOGPROCESS( spLogComp	 := MSG.COMP_RW, 
								spLogAction	 := MSG.ACTION_GET_MAGNET, 
								spLogStatus	 := MSG.STATUS_RUN,
								plogFlag	 := TRUE);
					process_G := 1;
					RETURN;
				END_IF
			ELSIF process_G = 1 THEN
//				KR1.PLC_O_D3.0 := TRUE; //200
				KR1.bOutBit[3,0] := TRUE;
				IF NOT KR1.bInBit[3,0] THEN
//					KR1.PLC_O_D3.0 := FALSE; //200	
					KR1.bOutBit[3,0] := FALSE;
					AUTO_MODE.processnameCOSMO := CONCAT(MSG.COMP_RW,MSG.ACTION_GET_MAGNET);
					AUTO_MODE.processnameCOSMO := CONCAT(AUTO_MODE.processnameCOSMO,MSG.STATUS_ACK);
					LOGPROCESS( spLogComp	 := MSG.COMP_RW, 
								spLogAction	 := MSG.ACTION_GET_MAGNET, 
								spLogStatus	 := MSG.STATUS_ACK,
								plogFlag	 := TRUE);
					process_G := 2;
					RETURN;
				END_IF	
			ELSIF process_G = 2 THEN
//				KR1.PLC_O_D3.0 := FALSE; //200	
				KR1.bOutBit[3,0] := FALSE;
				IF KR1.bInBit[3,0] THEN
					AUTO_MODE.processnameCOSMO := CONCAT(MSG.COMP_RW,MSG.ACTION_GET_MAGNET);
					AUTO_MODE.processnameCOSMO := CONCAT(AUTO_MODE.processnameCOSMO,MSG.STATUS_DONE);
					LOGPROCESS( spLogComp	 := MSG.COMP_RW, 
								spLogAction	 := MSG.ACTION_GET_MAGNET, 
								spLogStatus	 := MSG.STATUS_DONE,
								plogFlag	 := TRUE);
					process_G:= 3;
					RETURN;
				END_IF	
			ELSIF process_G = 3 THEN
				IF KR1.Idle THEN
					AUTO_MODE.processnameCOSMO := CONCAT(MSG.COMP_RW,MSG.ACTION_GET_MAGNET);
					AUTO_MODE.processnameCOSMO := CONCAT(AUTO_MODE.processnameCOSMO,MSG.STATUS_COMP);
					LOGPROCESS( spLogComp	 := MSG.COMP_RW, 
								spLogAction	 := MSG.ACTION_GET_MAGNET, 
								spLogStatus	 := MSG.STATUS_COMP,
								plogFlag	 := TRUE);
					process_G := 4;
					RW_sequence := 2;
					AUTO_MODE.next_step := FALSE;
					GVL.KR1_EOAT_FILL := TRUE;
				END_IF
			END_IF
		ELSE
			RW_sequence := 2;
		END_IF
		
	// Conveyor to Pitstop -------------------------------------------------------------------------------------------------------------	
	2: 
		IF process_X = 0 THEN
			IF KR1.Idle AND NOT GVL.Rework_Empty THEN
//				KR1.PLC_O_D3.7 := TRUE; //206
				KR1.bOutBit[3,7] := TRUE;
				AUTO_MODE.processnameCOSMO := CONCAT(MSG.COMP_RW,MSG.ACTION_REWORK_IN);
				AUTO_MODE.processnameCOSMO := CONCAT(AUTO_MODE.processnameCOSMO,MSG.STATUS_RUN);
				LOGPROCESS( spLogComp	 := MSG.COMP_RW, 
							spLogAction	 := MSG.ACTION_REWORK_IN, 
							spLogStatus	 := MSG.STATUS_RUN,
							plogFlag	 := TRUE);
				process_X := 1;
				AUTO_MODE.RW_PACKING := TRUE;
				RETURN;
			END_IF
		ELSIF process_X = 1 THEN
//			KR1.PLC_O_D3.7 := TRUE; //206
			KR1.bOutBit[3,7] := TRUE;
			IF KR1.bInBit[3,7] THEN
//				KR1.PLC_O_D3.7 := FALSE; //206	
				KR1.bOutBit[3,7] := FALSE;
				AUTO_MODE.processnameCOSMO := CONCAT(MSG.COMP_RW,MSG.ACTION_REWORK_IN);
				AUTO_MODE.processnameCOSMO := CONCAT(AUTO_MODE.processnameCOSMO,MSG.STATUS_ACK);
				LOGPROCESS( spLogComp	 := MSG.COMP_RW, 
							spLogAction	 := MSG.ACTION_REWORK_IN, 
							spLogStatus	 := MSG.STATUS_ACK,
							plogFlag	 := TRUE);
				process_X := 2;
				RETURN;
			END_IF	
		ELSIF process_X = 2 THEN
//			KR1.PLC_O_D3.7 := FALSE; //206	
			KR1.bOutBit[3,7] := FALSE;
			IF NOT KR1.bInBit[3,7] THEN
				AUTO_MODE.processnameCOSMO := CONCAT(MSG.COMP_RW,MSG.ACTION_REWORK_IN);
				AUTO_MODE.processnameCOSMO := CONCAT(AUTO_MODE.processnameCOSMO,MSG.STATUS_DONE);
				LOGPROCESS( spLogComp	 := MSG.COMP_RW, 
							spLogAction	 := MSG.ACTION_REWORK_IN, 
							spLogStatus	 := MSG.STATUS_DONE,
							plogFlag	 := TRUE);
				process_X:= 3;
				RETURN;
			END_IF
		ELSIF process_X = 3 THEN
			IF KR1.Idle THEN
					AUTO_MODE.processnameCOSMO := CONCAT(MSG.COMP_RW,MSG.ACTION_REWORK_IN);
					AUTO_MODE.processnameCOSMO := CONCAT(AUTO_MODE.processnameCOSMO,MSG.STATUS_COMP);
					LOGPROCESS( spLogComp	 := MSG.COMP_RW, 
								spLogAction	 := MSG.ACTION_REWORK_IN, 
								spLogStatus	 := MSG.STATUS_COMP,
								plogFlag	 := TRUE);
					process_X := 4;
					RW_sequence := 3;
					AUTO_MODE.next_step := FALSE;
					AUTO_MODE.KR1_PITSTOP := TRUE;
				END_IF
		END_IF	
		
	3:
		RW_sequence := 0;
		AUTO_MODE.next_step := FALSE;
		AUTO_MODE.processnameRW := CONCAT(MSG.COMP_RW,MAIN.fb_TimeStamp.SystemTime);
		AUTO_MODE.processnameRW := CONCAT(AUTO_MODE.processnameRW,MSG.STATUS_END);
		LOGPROCESS( spLogComp	 := MSG.COMP_RW, 
					spLogAction	 := MSG.ACTION_REWORK_IN, 
					spLogStatus	 := MSG.STATUS_END,
					plogFlag	 := TRUE);
END_CASE

END_PROGRAM

// ---- POUs/Auto_Seq/SEQ_LYR_PD0.TcPOU
PROGRAM SEQ_LYR_PD0
VAR_INPUT
	LYRPD_sequence	: UINT;
END_VAR

VAR
	process_Y	: UINT; //FG A IN
	process_Z	: UINT; //Place to Basket A A
	process_G	: UINT; //KR5 Get Magnet
	process_H	: UINT; //KR5 Remove Magnet
	bit1		: UINT;
	bit2		: UINT;
	
	Timer		: TON;
	
	fb_RunLayerPad	: FB_RunLayerPad;
	MSG_Bskt	: STRING;
END_VAR

IF GVL.LAYERPAD0 THEN
	RETURN;
END_IF

IF GVL.Rework_Empty AND NOT AUTO_MODE.FG_PACKING THEN
	RETURN;
END_IF

IF GVL.COSMO_UNLOAD THEN
	RETURN;
END_IF

IF NOT AUTO_MODE.FG_PACKING THEN
	Timer (IN:= TRUE, PT := T#5S);
	fb_RunLayerPad(Execute := FALSE);
	IF NOT timer.Q THEN
		RETURN;
	END_IF
END_IF

CASE LYRPD_sequence OF
	// Init ------------------------------------------------------------------------------------------------------------------	
	0:
		AUTO_MODE.processnameFG := CONCAT(MSG.COMP_FG,MSG.ACTION_INIT);	
		LOGPROCESS( spLogComp	 := MSG.COMP_FG, 
		 			spLogAction	 := MSG.ACTION_INIT, 
		 			spLogStatus	 := MSG.STATUS_DONE,
	 	 		 	plogFlag	 := TRUE);
		process_Y	:= 0;
		process_Z	:= 0;
		process_G	:= 0; // get magnet
		process_H	:= 0;
		AUTO_MODE.FG_PACKING := TRUE;
		fb_RunLayerPad(Execute := FALSE);
		Timer (IN:= FALSE);
		LYRPD_sequence := 1;
	
	// Check Layer Pad insertion -------------------------------------------------------------------------------------------------------------	
	1:	
		IF GVL.Basket_A_Counter = 0 THEN
			fb_RunLayerPad(Basket := 1, Layer := 0, Execute := TRUE);
			IF fb_RunLayerPad.Complete THEN
				fb_RunLayerPad(Execute := FALSE);
				LYRPD_sequence := 3;
			ELSIF fb_RunLayerPad.Error THEN
				fb_RunLayerPad(Execute := FALSE);
				AUTO_MODE.Halt_Production := TRUE;
				LYRPD_sequence := 2;
			END_IF
		ELSE
			GVL.LAYERPAD0 := TRUE;
		END_IF
	
	3:
		LYRPD_sequence := 0;
		GVL.LAYERPAD0 := TRUE;
		AUTO_MODE.next_step := FALSE;
		AUTO_MODE.FG_PACKING := FALSE;
		AUTO_MODE.processnameFG := CONCAT(MSG.COMP_FG,MAIN.fb_TimeStamp.SystemTime);
		AUTO_MODE.processnameFG := CONCAT(AUTO_MODE.processnameFG,MSG.STATUS_END);
		LOGPROCESS( spLogComp	 := MSG.COMP_FG, 
					spLogAction	 := MSG.ACTION_FG_PACK, 
					spLogStatus	 := MSG.STATUS_END,
					plogFlag	 := TRUE);
END_CASE

END_PROGRAM

// ---- POUs/Auto_Seq/SEQ_FG.TcPOU
PROGRAM SEQ_FG
VAR_INPUT
	FG_sequence	: UINT;
END_VAR

VAR
	process_Y	: UINT; //Pitstop to Basket B
	process_Z	: UINT; //Pitstop to Basket A
	process_G	: UINT; //KR1 GET Magnet
	process_H	: UINT; //KR1 Remove Magnet
	
END_VAR


IF NOT AUTO_MODE.KR1_PITSTOP THEN
	RETURN;
END_IF

CASE FG_sequence OF
	0:
		AUTO_MODE.processnameFG := CONCAT(MSG.COMP_FG,MSG.ACTION_INIT);	
		LOGPROCESS( spLogComp	 := MSG.COMP_FG, 
		 			spLogAction	 := MSG.ACTION_INIT, 
		 			spLogStatus	 := MSG.STATUS_DONE,
	 	 		 	plogFlag	 := TRUE);
		process_Y	:= 0;
		process_Z	:= 0;
		process_G	:= 0;
		process_H	:= 0;
		AUTO_MODE.FG_PACKING := TRUE;
		FG_sequence := 1;
	
	// Pitstop to Basket -------------------------------------------------------------------------------------------------------------	
	1:
		IF process_Z = 0 THEN
			CASE GVL.Basket_A_Counter OF
				0:
//					KR1.bOutBit[2,0] := TRUE;
//					KR1.PLC_O_D4.2 := TRUE; //208
					KR1.bOutBit[4,2] := TRUE;
					AUTO_MODE.processnameFG := CONCAT(MSG.COMP_FG,MSG.ACTION_FGA_POS1);
					AUTO_MODE.processnameFG := CONCAT(AUTO_MODE.processnameFG,MSG.STATUS_RUN);
					LOGPROCESS( spLogComp	 := MSG.COMP_FG, 
								spLogAction	 := MSG.ACTION_FGA_POS1, 
								spLogStatus	 := MSG.STATUS_RUN,
								plogFlag	 := TRUE);
					process_Z := 1;
					RETURN;
				1:
//					KR1.bOutBit[2,1] := TRUE;
//					KR1.PLC_O_D4.3 := TRUE; //209
					KR1.bOutBit[4,3] := TRUE;
					AUTO_MODE.processnameFG := CONCAT(MSG.COMP_FG,MSG.ACTION_FGA_POS2);
					AUTO_MODE.processnameFG := CONCAT(AUTO_MODE.processnameFG,MSG.STATUS_RUN);
					LOGPROCESS( spLogComp	 := MSG.COMP_FG, 
								spLogAction	 := MSG.ACTION_FGA_POS2, 
								spLogStatus	 := MSG.STATUS_RUN,
								plogFlag	 := TRUE);
					process_Z := 1;
					RETURN;
				2:
//					KR1.bOutBit[2,2] := TRUE;
//					KR1.PLC_O_D4.4 := TRUE; //210
					KR1.bOutBit[4,4] := TRUE;
					AUTO_MODE.processnameFG := CONCAT(MSG.COMP_FG,MSG.ACTION_FGA_POS3);
					AUTO_MODE.processnameFG := CONCAT(AUTO_MODE.processnameFG,MSG.STATUS_RUN);
					LOGPROCESS( spLogComp	 := MSG.COMP_FG, 
								spLogAction	 := MSG.ACTION_FGA_POS3, 
								spLogStatus	 := MSG.STATUS_RUN,
								plogFlag	 := TRUE);
					process_Z := 1;
					RETURN;
				3:
//					KR1.bOutBit[2,3] := TRUE;
//					KR1.PLC_O_D4.5 := TRUE; //211
					KR1.bOutBit[4,5] := TRUE;
					AUTO_MODE.processnameFG := CONCAT(MSG.COMP_FG,MSG.ACTION_FGA_POS4);
					AUTO_MODE.processnameFG := CONCAT(AUTO_MODE.processnameFG,MSG.STATUS_RUN);
					LOGPROCESS( spLogComp	 := MSG.COMP_FG, 
								spLogAction	 := MSG.ACTION_FGA_POS4, 
								spLogStatus	 := MSG.STATUS_RUN,
								plogFlag	 := TRUE);
					process_Z := 1;
					RETURN;
				4:
//					KR1.bOutBit[2,4] := TRUE;
//					KR1.PLC_O_D4.6 := TRUE; //212
					KR1.bOutBit[4,6] := TRUE;
					AUTO_MODE.processnameFG := CONCAT(MSG.COMP_FG,MSG.ACTION_FGA_POS5);
					AUTO_MODE.processnameFG := CONCAT(AUTO_MODE.processnameFG,MSG.STATUS_RUN);
					LOGPROCESS( spLogComp	 := MSG.COMP_FG, 
								spLogAction	 := MSG.ACTION_FGA_POS5, 
								spLogStatus	 := MSG.STATUS_RUN,
								plogFlag	 := TRUE);
					process_Z := 1;
					RETURN;
			END_CASE
		ELSIF process_Z = 1 THEN
			IF KR1.PLC_I_PROG1 <> 0 THEN
				KR1.PLC_O_PROG1 := 0; //208-215	
				AUTO_MODE.processnameFG := CONCAT(MSG.COMP_FG,MSG.ACTION_FGA_POS);
				AUTO_MODE.processnameFG := CONCAT(AUTO_MODE.processnameFG,MSG.STATUS_ACK);
				LOGPROCESS( spLogComp	 := MSG.COMP_FG, 
							spLogAction	 := MSG.ACTION_FGA_POS, 
							spLogStatus	 := MSG.STATUS_ACK,
							plogFlag	 := TRUE);
				process_Z := 2;
				RETURN;
			END_IF	
		ELSIF process_Z = 2 THEN
			IF KR1.PLC_O_PROG1 = 0 THEN
				AUTO_MODE.processnameFG := CONCAT(MSG.COMP_FG,MSG.ACTION_FGA_POS);
				AUTO_MODE.processnameFG := CONCAT(AUTO_MODE.processnameFG,MSG.STATUS_DONE);
				LOGPROCESS( spLogComp	 := MSG.COMP_FG, 
							spLogAction	 := MSG.ACTION_FGA_POS, 
							spLogStatus	 := MSG.STATUS_DONE,
							plogFlag	 := TRUE);
				process_Z:= 3;
				GVL.daily_output := GVL.daily_output+1;
				GVL.weekly_output := GVL.weekly_output+1;
				GVL.monthly_output := GVL.monthly_output+1;
				IF AUTO_MODE.RW_PACKING THEN
					GVL.Rework_Counter := GVL.Rework_Counter+1;
				ELSE
					GVL.Pass_Counter := GVL.Pass_Counter+1;
				END_IF
				
				IF GVL.Basket_A_Counter < 4 THEN
					GVL.Basket_A_Counter := GVL.Basket_A_Counter+1;
				ELSE
					GVL.Basket_A_Counter := 0;
				END_IF
				
				FG_sequence := 2;
				AUTO_MODE.next_step := FALSE;
				AUTO_MODE.KR1_PITSTOP := FALSE;
				AUTO_MODE.FG_PACKING := FALSE;
				AUTO_MODE.RW_PACKING := FALSE;
				AUTO_MODE.processnameFG := CONCAT(MSG.COMP_FG,MSG.ACTION_FGA_POS);
				AUTO_MODE.processnameFG := CONCAT(AUTO_MODE.processnameFG,MSG.STATUS_COMP);
				LOGPROCESS( spLogComp	 := MSG.COMP_FG, 
							spLogAction	 := MSG.ACTION_FGA_POS, 
							spLogStatus	 := MSG.STATUS_COMP,
							plogFlag	 := TRUE);
			END_IF	
		END_IF
		
	2:
		FG_sequence := 0;
		AUTO_MODE.next_step := FALSE;
		AUTO_MODE.KR1_PITSTOP := FALSE;
		AUTO_MODE.processnameFG := CONCAT(MSG.COMP_FG,MAIN.fb_TimeStamp.SystemTime);
		AUTO_MODE.processnameFG := CONCAT(AUTO_MODE.processnameFG,MSG.STATUS_END);
		LOGPROCESS( spLogComp	 := MSG.COMP_FG, 
					spLogAction	 := MSG.ACTION_FG_PACK, 
					spLogStatus	 := MSG.STATUS_END,
					plogFlag	 := TRUE);
END_CASE

END_PROGRAM

// ---- POUs/LOGGING/LOGFILE.TcPOU
PROGRAM LOGFILE
VAR_INPUT
	sLogEvent	: STRING;
	sLogComp	: STRING;
	sLogAction	: STRING;
//	sLogStatus	: STRING;
	logFlag		: bool;
END_VAR
VAR_OUTPUT
	log_complete : BOOL := FALSE;
	log_error	 : BOOL := FALSE;
END_VAR
VAR
	fb_TimeStamp : FB_UpdateTimeStamp ();
	fbCreateDir	 : FB_CreateDir;
	fbFileOpen	 : FB_FileOpen;
	fbFileWrite	 : FB_FilePuts;
	fbFileClose	 : FB_FileClose;
	log_state	 : (	INIT, 
					 CREATE_DIR, 
					 FILE_OPEN,
					 WRITE_TITLE,
					 WRITE_LOG, 
					 FILE_CLOSE,
					 CLEAR, 
					 ERROR);
					
	writeLog	 : STRING[255];
	writeTitle	 : STRING;
	sFolderName	 : STRING;
	swFolderName	 : STRING;
	sFileName	 : STRING;
	sTextLog	 : STRING;
	swTextLog	 : STRING;
	lastFileName : STRING;	
	swLogEvent	: STRING;
	swLogComp	: STRING;
	swLogAction	: STRING;
	swLogStatus	: STRING;
	
END_VAR

//IF sLogEvent<>swLogEvent OR sLogComp<>swLogComp OR sLogAction<>swLogAction THEN
//	swLogEvent	:= sLogEvent;
//	swLogComp	:= sLogComp;
//	swLogAction	:= sLogAction;
////	swLogStatus	:= sLogStatus;
//ELSE
//	RETURN;
//END_IF

sTextLog := str_concat(sLogEvent,sLogComp,sLogAction);

WHILE logFlag DO
	CASE log_state OF
		// INIT -------------------------------------------------------------------
		INIT:
			log_complete	:= FALSE;
			log_error		:= FALSE;
			log_state 		:= CREATE_DIR;
			fbCreateDir(bExecute:= FALSE);
	
		// CREATE_DIR -------------------------------------------------------------			
		CREATE_DIR:	
			sFolderName := CONCAT('C:\Users\Administrator\Desktop\log\HMI\', MAIN.fb_TimeStamp.SystemDate);
//			sFolderName := CONCAT('C:\Users\celli\OneDrive\Desktop\YISB_LOG\HMI\', MAIN.fb_TimeStamp.SystemDate);

			IF sFolderName = swFolderName THEN
				log_state := FILE_OPEN;
				fbCreateDir(bExecute := FALSE);
				fbFileOpen(bExecute := FALSE);
			ELSE
				fbCreateDir( sPathName:= sFolderName, bExecute:= TRUE );
				IF NOT fbCreateDir.bBusy THEN
					log_state := FILE_OPEN;
					fbCreateDir(bExecute := FALSE);
					fbFileOpen(bExecute := FALSE);
					swFolderName := sFolderName;
				END_IF
			END_IF
			
		// FILE_OPEN -------------------------------------------------------------
		FILE_OPEN:
			sFileName := CONCAT(sFolderName,'\');
			sFileName := CONCAT(sFileName, MAIN.fb_TimeStamp.SystemHour);
			sFileName := CONCAT(sFileName,'.csv');
				
			fbFileOpen( sPathName:= sFileName, 
						nMode:= FOPEN_MODEAPPEND, 
						bExecute:= TRUE, 
						hFile=>);
			IF fbFileOpen.bError THEN
				log_state := ERROR;
				fbFileOpen(bExecute := FALSE);
				fbFileWrite(bExecute := FALSE);
			ELSIF NOT fbFileOpen.bBusy THEN
				log_state := WRITE_TITLE;
				fbFileOpen(bExecute := FALSE);
				fbFileWrite(bExecute := FALSE);
			END_IF
			
		// WRITE_TITLE -------------------------------------------------------------
		WRITE_TITLE:
			IF lastFileName <> sFileName THEN	
				writeTitle := CONCAT('$n','Time Stamp');
				writeTitle := CONCAT(writeTitle,';');
				writeTitle := CONCAT(writeTitle,'Event');
				writeTitle := CONCAT(writeTitle,';');
				writeTitle := CONCAT(writeTitle,'Component');
				writeTitle := CONCAT(writeTitle,';');
				writeTitle := CONCAT(writeTitle,'Action');
				
				fbFileWrite ( hFile:=fbFileOpen.hFile,
								sLine:=writeTitle,
								bExecute:=TRUE);
				IF fbFileWrite.bError THEN
					log_state := ERROR;
					fbFileWrite(bExecute := FALSE);
					fbFileClose(bExecute := FALSE);
				ELSIF NOT fbFileWrite.bBusy THEN
					log_state := WRITE_LOG;
					fbFileWrite(bExecute := FALSE);
					fbFileClose(bExecute := FALSE);
					lastFileName := sFileName;
				END_IF
			ELSE
				log_state := WRITE_LOG;
			END_IF

		// WRITE_LOG -------------------------------------------------------------
		WRITE_LOG:	
			writeLog := sTextLog;
			
			fbFileWrite ( hFile:=fbFileOpen.hFile,
							sLine:=writeLog,
							bExecute:=TRUE);
			IF fbFileWrite.bError THEN
				log_state := ERROR;
				fbFileWrite(bExecute := FALSE);
				fbFileClose(bExecute := FALSE);
			ELSIF NOT fbFileWrite.bBusy THEN
				log_state := FILE_CLOSE;
				fbFileWrite(bExecute := FALSE);
				fbFileClose(bExecute := FALSE);
			END_IF
			
		// FILE_CLOSE -------------------------------------------------------------
		FILE_CLOSE:			
			fbFileClose( hFile:=fbFileOpen.hFile,
						 bExecute:=TRUE);
			IF fbFileClose.bError THEN
				log_state := ERROR;
				fbFileClose(bExecute := FALSE);
			ELSIF NOT fbFileClose.bBusy THEN
				log_state := CLEAR;
				fbFileClose(bExecute := FALSE);
			END_IF
			
		// CLEAR -------------------------------------------------------------	
		CLEAR:
			log_complete	:= TRUE;
			logFlag			:= FALSE;
			log_state 		:= INIT;
				
		// ERROR -------------------------------------------------------------	
		ERROR:
			log_error		:= TRUE;
			logFlag			:= FALSE;
			log_state 		:= INIT;
	END_CASE
END_WHILE

METHOD str_concat : STRING
VAR_INPUT
	text1	: STRING;
	text2	: STRING;
	text3	: STRING;
//	text4	: STRING;
END_VAR
VAR
	Con_String : String;
END_VAR
Con_String := CONCAT('$n', MAIN.fb_TimeStamp.FullSystemTime);
Con_String := CONCAT(Con_String, ' ; ');
Con_String := CONCAT(Con_String, text1);
Con_String := CONCAT(Con_String, ' ; ');
Con_String := CONCAT(Con_String, text2);
Con_String := CONCAT(Con_String, ' ; ');
Con_String := CONCAT(Con_String, text3);
//Con_String := CONCAT(Con_String, ' ; ');
//Con_String := CONCAT(Con_String, text4);

str_concat := Con_String;
END_METHOD

END_PROGRAM

// ---- POUs/Kuka IO/KUKA_IO.TcPOU
PROGRAM KUKA_IO
VAR_INPUT
	LogText : STRING;
END_VAR

KR1();
KR2();
KR3();
KR4();
KR5();

END_PROGRAM

// ---- POUs/JIG.TcPOU
PROGRAM JIG
VAR
	BasketA_Plus	: BOOL;
	BasketA_Minus	: BOOL;
	BasketB_Plus	: BOOL;
	BasketB_Minus	: BOOL;
	MAX_FG_ON_BASKET : UINT := 15;
END_VAR

IF AUTO_MODE.AutoMode THEN
	RETURN;
END_IF

GVL.JIGA_Release := NOT GVL.JIGA_Clamp;
GVL.JIGB_Release := NOT GVL.JIGB_Clamp;
GVL.JIGC_Release := NOT GVL.JIGC_Clamp;

IF BasketA_Plus THEN
	GVL.Basket_A_Counter := GVL.Basket_A_Counter + 1;
	IF GVL.Basket_A_Counter > MAX_FG_ON_BASKET THEN
		GVL.Basket_A_Counter := 0 ;
	END_IF
	BasketA_Plus := FALSE;
END_IF

IF BasketA_Minus THEN
	GVL.Basket_A_Counter := GVL.Basket_A_Counter - 1;
	IF GVL.Basket_A_Counter < 0 THEN
		GVL.Basket_A_Counter := MAX_FG_ON_BASKET;
	END_IF
	BasketA_Minus := FALSE;
END_IF

IF BasketB_Plus THEN
	GVL.Basket_B_Counter := GVL.Basket_B_Counter + 1;
	IF GVL.Basket_B_Counter > MAX_FG_ON_BASKET THEN
		GVL.Basket_B_Counter := 0 ;
	END_IF
	BasketB_Plus := FALSE;
END_IF

IF BasketB_Minus THEN
	GVL.Basket_B_Counter := GVL.Basket_B_Counter - 1;
	IF GVL.Basket_B_Counter < 0 THEN
		GVL.Basket_B_Counter := MAX_FG_ON_BASKET;
	END_IF
	BasketB_Minus := FALSE;
END_IF

END_PROGRAM

// ---- POUs/SAFETY_SENSOR.TcPOU
PROGRAM SAFETY_SENSOR
VAR_INPUT
	safety_compromised : BOOL;
	WELDING_MODE : BOOL;
END_VAR
VAR
	SENSOR_AIR_PRESSURE_OK AT %I* : BOOL;
	SENSOR_GAS_PRESSURE_OK AT %I* : BOOL;
	SENSOR_AIR_PRESSURE_HIGH AT %I* : BOOL;
	SENSOR_GAS_PRESSURE_HIGH AT %I* : BOOL;
	SENSOR_SAFETY_DOOR_CLOSE AT %I* : BOOL;
	
END_VAR


IF AUTO_MODE.AutoMode THEN	
	IF	NOT SENSOR_SAFETY_DOOR_CLOSE OR
		NOT SENSOR_AIR_PRESSURE_OK OR 
		SENSOR_AIR_PRESSURE_HIGH THEN 
			safety_compromised := TRUE;
			KR1.bOutBit[1,0]:= FALSE;
			KR2.bOutBit[1,0]:= FALSE;
			KR3.bOutBit[1,0]:= FALSE;
			KR4.bOutBit[1,0]:= FALSE;
			KR5.bOutBit[1,0]:= FALSE;
			AUTO_MODE.Halt_Production := TRUE;
			AUTO_MODE.AutoMode := FALSE;
	ELSIF WELDING_MODE THEN
		IF  NOT SENSOR_AIR_PRESSURE_OK OR 
			NOT SENSOR_GAS_PRESSURE_OK OR
			SENSOR_AIR_PRESSURE_HIGH OR
			SENSOR_GAS_PRESSURE_HIGH OR 
			NOT SENSOR_SAFETY_DOOR_CLOSE THEN
				KR1.bOutBit[1,0]:= FALSE;
				KR2.bOutBit[1,0]:= FALSE;
				KR3.bOutBit[1,0]:= FALSE;
				KR4.bOutBit[1,0]:= FALSE;
				KR5.bOutBit[1,0]:= FALSE;
				safety_compromised := TRUE;
				AUTO_MODE.Halt_Production := TRUE;
				AUTO_MODE.AutoMode := FALSE;
		ELSE
			safety_compromised := FALSE;		
		END_IF
	ELSE
		safety_compromised := FALSE;
	END_IF
ELSE
	IF	NOT SENSOR_SAFETY_DOOR_CLOSE OR
		NOT SENSOR_AIR_PRESSURE_OK OR 
		SENSOR_AIR_PRESSURE_HIGH THEN 
			safety_compromised := TRUE;
	ELSIF WELDING_MODE THEN
		IF  NOT SENSOR_AIR_PRESSURE_OK OR 
			NOT SENSOR_GAS_PRESSURE_OK OR
			SENSOR_AIR_PRESSURE_HIGH OR
			SENSOR_GAS_PRESSURE_HIGH OR 
			NOT SENSOR_SAFETY_DOOR_CLOSE THEN
				safety_compromised := TRUE;
		ELSE
			safety_compromised := FALSE;		
		END_IF
	ELSE
		safety_compromised := FALSE;
	END_IF
	
END_IF

END_PROGRAM

// ---- POUs/TL.TcPOU
PROGRAM TL
VAR_INPUT
	TL_Green	AT %Q* : BOOL;
	TL_Ember	AT %Q* : BOOL;
	TL_Red		AT %Q* : BOOL;
	TL_Buzzer	AT %Q* : BOOL;
END_VAR
VAR
	tOn 	: TON;
	tOff 	: TON;
	bOn		: BOOL;
	blastOn	: BOOL;
	Buzzer_mute: BOOL := TRUE;
END_VAR


TL_Ember := KR1.KR_ProgReady AND KR2.KR_ProgReady AND KR3.KR_ProgReady AND KR4.KR_ProgReady AND KR5.KR_ProgReady;
TL_Green := AUTO_MODE.AutoMode AND NOT TL_Red;

IF NOT MAIN.btnEstop OR MAIN.btnSoftEstop OR SAFETY_SENSOR.safety_compromised THEN
	tOn(IN:= NOT tOff.Q, PT:= T#1S, Q=> bOn , ET=> );
	tOff(IN:= bOn, PT:= T#0.5S, Q=> , ET=> );
	
	TL_Red := bOn;
	IF Buzzer_mute THEN
		TL_Buzzer := FALSE;
	ELSE
		TL_Buzzer := bOn;
	END_IF
ELSIF AUTO_MODE.AutoMode THEN
	IF NOT KR1.KR_ProgReady OR NOT KR2.KR_ProgReady OR NOT KR3.KR_ProgReady OR NOT KR4.KR_ProgReady OR NOT KR5.KR_ProgReady OR 
		AUTO_MODE.JIGA_ErrorState OR AUTO_MODE.JIGB_ErrorState OR AUTO_MODE.JIGC_ErrorState OR AUTO_MODE.TT_ErrorState 
		THEN
			tOn(IN:= NOT tOff.Q, PT:= T#0.5S, Q=> bOn , ET=> );
			tOff(IN:= bOn, PT:= T#0.5S, Q=> , ET=> );
		
			TL_Red := bOn;
			IF Buzzer_mute THEN
				TL_Buzzer := FALSE;
			ELSE
				TL_Buzzer := bOn;
			END_IF
	ELSE
		TL_Buzzer := TL_Red := FALSE;
	END_IF
ELSE
	TL_Buzzer := TL_Red := FALSE;
END_IF

END_PROGRAM

// ---- POUs/TORCHCLEAN.TcPOU
PROGRAM TORCHCLEAN
VAR_INPUT
	KR_TC	: BOOL;
	process_A	: INT;
END_VAR
VAR
	TC_sequence	: INT;
END_VAR


CASE TC_sequence OF
	0:
		IF process_A = 0 THEN
			IF KR1.Idle AND KR2.Idle AND KR3.Idle AND KR4.Idle THEN
				KR3.bOutBit[3,2]:= TRUE; //302
				KR4.bOutBit[3,1] := TRUE; //301
				KR_TC := TRUE;
				process_A := 1;
				RETURN;
			END_IF
		ELSIF process_A = 1 THEN
			IF KR3.bInBit[3,2] AND KR4.bInBit[3,1] THEN
				KR3.bOutBit[3,2]:= FALSE; //302
				KR4.bOutBit[3,1] := FALSE; //301
				process_A := 2;
				RETURN;
			END_IF	
		ELSIF process_A = 2 THEN
			IF NOT KR3.bInBit[3,2] AND NOT KR4.bInBit[3,1] THEN
				process_A:= 3;
				RETURN;
			END_IF	
		ELSIF process_A = 3 THEN
			IF KR3.Idle AND KR4.Idle THEN
				KR_TC := FALSE;
				MAIN.btnTorchClean := FALSE;
				process_A := 0;
				TC_sequence := 0;
			END_IF
		END_IF
END_CASE

END_PROGRAM

// ---- POUs/LOGGING.TcPOU
PROGRAM LOGGING
VAR_INPUT
	sWriteLog		: STRING[255];
	sLog			: STRING[255];
//	dir_log 		: UINT;
	bLogFlag		: BOOL;
	LogState		: INT;
END_VAR
VAR_OUTPUT
	bError				: BOOL;
	nErrID				: UDINT;
END_VAR
VAR
	CreateDir	: FB_CreateDir;
	FileOpen	: FB_FileOpen;
	FileWrite	: FB_FileWrite;
	FileClose	: FB_FileClose;
	
    ePath        	: E_OpenPath; (* folders root path *)
    sPathName     	: STRING;
	bBootFolder		: BOOL;
	writeBuffer		: STRING[255] := '';
	hfile			: UINT;
	
	sTxtName	: T_MaxString;
	sFolderName	: T_MaxString;
	DirCreateError	: BOOL;
	FileOpenError	: BOOL;
	FileWriteError	: BOOL;
	FileCloseError	: BOOL;
	sTimeStamp: STRING(255);
	
	writeFlag		: BOOL;
	lastLog			: String[255];
END_VAR

IF sLog = lastLog THEN
	RETURN;
END_IF

//CASE LogState OF
//	0:
//		writeFlag := TRUE;
//		// Set Log Folder Name
////		sFolderName := CONCAT ('C:\Users\celli\OneDrive\Desktop\YISB_LOG\',LOG_TIME_STAMP.Local_Date);
//		sFolderName := CONCAT ('C:\Users\Administrator\Desktop\log\',LOG_TIME_STAMP.Local_Date);
		
//		CreateDir(
//				sNetId:= '', 
//				sPathName:= sFolderName, 
//				ePath:= PATH_GENERIC, 
//				bExecute:= TRUE, 
//				tTimeout:= DEFAULT_ADS_TIMEOUT, 
//				bBusy=> , 
//				bError=> DirCreateError, 
//				nErrId=> nErrID);
//			IF CreateDir.tTimeout > DEFAULT_ADS_TIMEOUT THEN
//				LogState := 0;
//				bLogFlag := FALSE;
//				CreateDir.bExecute := FALSE;
//				FileOpen(bExecute := FALSE);
//				MAIN.BTN_LOG := FALSE;
//				RETURN;
//			ELSIF NOT CreateDir.bBusy THEN
//				LogState := 1;
//				CreateDir.bExecute := FALSE;
//				FileOpen(bExecute := FALSE);
//			END_IF

//		// Open File	
//		1:
//			// Set Log File Name	
//			sTxtName := WORD_TO_STRING(LOG_TIME_STAMP.LocalTime.systemTime.wHour);
//			sTxtName := CONCAT(sTxtName, '.txt');
//			sTxtName := CONCAT('\',sTxtName,);
//			sTxtName := CONCAT(sFolderName,sTxtName);
			
//			FileOpen(
//				sNetId:= , 
//				sPathName:= sTxtName, 
//				nMode:= FOPEN_MODEAPPEND, 
//				ePath:= PATH_GENERIC, 
//				bExecute:= TRUE, 
//				tTimeout:= DEFAULT_ADS_TIMEOUT, 
//				bBusy=> , 
//				bError=> FileOpenError, 
//				nErrId=> nErrID, 
//				hFile=> hfile);
//			IF FileOpenError OR FileOpen.tTimeout > DEFAULT_ADS_TIMEOUT THEN
//				LogState := 0;
//				bLogFlag := FALSE;
//				FileOpen.bExecute := FALSE;
//				FileWrite(bExecute := FALSE);
//				MAIN.BTN_LOG := FALSE;
//				RETURN;
//			ELSIF NOT FileOpen.bBusy THEN
//				LogState := 2;
//				FileOpen.bExecute := FALSE;
//				FileWrite(bExecute := FALSE);
//			END_IF
			
//		// Write File
//		2:	
//				// Set Log messages	
//				sTimeStamp 	:= CONCAT('$n',SYSTEMTIME_TO_STRING(LOG_TIME_STAMP.LocalTime.systemTime));
//				sTimeStamp 	:= CONCAT(sTimeStamp,' - ');
//				sWriteLog 	:= CONCAT(sTimeStamp, sLog);
//				writeBuffer := sWriteLog;
				
//				FileWrite(
//					sNetId:= , 
//					hFile:= hfile, 
//					pWriteBuff:= ADR(writeBuffer), 
//					cbWriteLen:= INT_TO_UDINT(LEN(writeBuffer)), 
//					bExecute:= TRUE, 
//					tTimeout:= T#3S, 
//					bBusy=> , 
//					bError=> FileWriteError, 
//					nErrId=> nErrID, 
//					cbWrite=> );
					
//			IF FileWriteError OR FileWrite.tTimeout > DEFAULT_ADS_TIMEOUT THEN
//				LogState := 0;
//				bLogFlag := FALSE;
//				FileWrite.bExecute := FALSE;
//				MAIN.BTN_LOG := FALSE;
//				writeFlag:= FALSE;
//				FileClose(bExecute := FALSE);
//				RETURN;
//			ELSIF NOT FileWrite.bBusy THEN
//				LogState := 3;
//				writeFlag:= FALSE;
//				FileWrite.bExecute := FALSE;
//				FileClose(bExecute := FALSE);
//			END_IF
			
//		// Close File
//		3:
//			FileClose(
//				sNetId:= , 
//				hFile:= hfile, 
//				bExecute:= TRUE,
//				tTimeout:= T#3S, 
//				bBusy=> , 
//				bError=> FileCloseError, 
//				nErrId=> nErrID);
//			IF FileCloseError OR FileClose.tTimeout > DEFAULT_ADS_TIMEOUT THEN
//				LogState := 0;
//				bLogFlag := FALSE;
//				lastLog := sLog;
//				FileClose(bExecute := FALSE);
//				MAIN.BTN_LOG := FALSE;
//				RETURN;
//			ELSIF NOT FileClose.bBusy THEN
//				LogState := 0;
//				lastLog := sLog;
//				FileClose(bExecute := FALSE);
//				CreateDir(bExecute:= FALSE);
//				bLogFlag := FALSE;
//				MAIN.BTN_LOG := FALSE;
//			END_IF
//END_CASE

END_PROGRAM

// ---- POUs/LOG_TIME_STAMP.TcPOU
PROGRAM LOG_TIME_STAMP
VAR
END_VAR
VAR_INPUT
	LocalTime: FB_LocalSystemTime;
	Local_Date	: STRING;
	Local_Time	: STRING;
END_VAR



//================================ Function Block

LocalTime(
		sNetID:= , 
		bEnable:= TRUE , 
		dwCycle:= 1, 
		dwOpt:= , 
		tTimeout:= ,
		bValid=> , 
		systemTime=> , 
		tzID=> );

//================================ Footer System Time

IF NOT LocalTime.bValid THEN
	RETURN;
END_IF
		
Local_Date := CONCAT (WORD_TO_STRING(LocalTime.systemTime.wYear),' - ');
Local_Date := CONCAT (Local_Date, WORD_TO_STRING(LocalTime.systemTime.wMonth));
Local_Date := CONCAT (Local_Date, ' - ');
Local_Date := CONCAT (Local_Date, WORD_TO_STRING(LocalTime.systemTime.wDay));

Local_Time := CONCAT (WORD_TO_STRING(LocalTime.systemTime.wHour),' : ');
Local_Time := CONCAT (Local_Time, WORD_TO_STRING(LocalTime.systemTime.wMinute));
Local_Time := CONCAT (Local_Time, ' : ');
Local_Time := CONCAT (Local_Time, WORD_TO_STRING(LocalTime.systemTime.wSecond));

END_PROGRAM

